Fanuc TP program (LS listing): MAKROSTP.LS

/PROG  MAKROSTP
/ATTR
OWNER		= MNEDITOR;
COMMENT		= "MAKRO_SCHRITT";
PROG_SIZE	= 100704;
CREATE		= DATE 11-01-11  TIME 07:00:00;
MODIFIED	= DATE 18-12-28  TIME 09:20:00;
FILE_NAME	= ;
VERSION		= 0;
LINE_COUNT	= 4405;
MEMORY_SIZE	= 103104;
PROTECT		= READ_WRITE;
TCD:  STACK_SIZE	= 0,
      TASK_PRIORITY	= 100,
      TIME_SLICE	= 0,
      BUSY_LAMP_OFF	= 1,
      ABORT_REQUEST	= 7,
      PAUSE_REQUEST	= 3;
DEFAULT_GROUP	= *,*,*,*,*;
CONTROL_CODE	= 00000000 00000010;
/MN
    :  !Schrittkette Konzernstandard ;
    :  !KS24 ;
    :  !Version: 02 ;
    :  !Stand: 003 MOD KN ;
    :  !letzte Aenderung 30.07.2015 DB ;
    :  !Mod von KN --> S2 mit Wartezeit ;
    :   ;
    :  !Zaehler [41] = aktueller Schritt ;
    :  !Zaehler [42] = letzter Schritt ;
    :  R[41]=0    ;
    :  R[42]=0    ;
    :   ;
    :   ;
    :  !*********************** ;
    :  !*********************** ;
    :  !* Start Makro_Schritt * ;
    :  !*********************** ;
    :  !*********************** ;
    :   ;
    :   ;
    :  !***************************** ;
    :  !*         Schritt 1         * ;
    :  !* E/A's / Flags Ruecksetzen * ;
    :  !***************************** ;
    :   ;
    :  !Loop fuer Schrittkette LBL[1] ;
    :  LBL[1] ;
    :  R[41]=1    ;
    :  !Statusbildschirm einblenden ;
    :  DO[18181]=(OFF) ;
    :  !SK1 KF1 KS1 ;
    :  DO[786]=(OFF) ;
    :  DO[834]=(OFF) ;
    :  DO[842]=(OFF) ;
    :  DO[847]=(OFF) ;
    :  !SK2 KF2 KS2 ;
    :  DO[946]=(OFF) ;
    :  DO[994]=(OFF) ;
    :  DO[995]=(OFF) ;
    :  DO[1002]=(OFF) ;
    :  !SK3 KF3 KS3 ;
    :  DO[1106]=(OFF) ;
    :  DO[1154]=(OFF) ;
    :  DO[1155]=(OFF) ;
    :  DO[1162]=(OFF) ;
    :  !KS1 KS2 KS3 ;
    :  DO[3969]=(OFF) ;
    :  DO[3970]=(OFF) ;
    :  DO[3971]=(OFF) ;
    :  !Auswahl EZ1/SP1 an KF2 ;
    :  F[72]=(OFF) ;
    :  !Auswahl EZ1/SP1 an KF3 ;
    :  F[73]=(OFF) ;
    :  !Auswert. KF Umdrehungen EZ1/SP1 ;
    :  F[94]=(OFF) ;
    :  F[95]=(OFF) ;
    :  F[96]=(OFF) ;
    :  F[97]=(OFF) ;
    :  F[98]=(OFF) ;
    :  F[99]=(OFF) ;
    :  F[100]=(OFF) ;
    :  F[101]=(OFF) ;
    :  F[102]=(OFF) ;
    :  F[103]=(OFF) ;
    :  F[104]=(OFF) ;
    :  F[105]=(OFF) ;
    :  F[106]=(OFF) ;
    :  F[107]=(OFF) ;
    :  F[108]=(OFF) ;
    :  F[109]=(OFF) ;
    :  F[110]=(OFF) ;
    :  F[111]=(OFF) ;
    :  F[112]=(OFF) ;
    :  F[113]=(OFF) ;
    :  F[114]=(OFF) ;
    :  F[115]=(OFF) ;
    :  F[116]=(OFF) ;
    :  F[117]=(OFF) ;
    :  !Auswert. KF Umdrehungen EZ2/SP2 ;
    :  F[150]=(OFF) ;
    :  F[151]=(OFF) ;
    :  F[152]=(OFF) ;
    :  F[153]=(OFF) ;
    :  F[154]=(OFF) ;
    :  F[155]=(OFF) ;
    :  !Auswert. KF Umdrehungen EZ3/SP3 ;
    :  F[186]=(OFF) ;
    :  F[187]=(OFF) ;
    :  F[188]=(OFF) ;
    :  F[189]=(OFF) ;
    :  F[190]=(OFF) ;
    :  F[191]=(OFF) ;
    :  !Hilfsflags beim Fraesen ;
    :  F[287]=(OFF) ;
    :  F[290]=(OFF) ;
    :  F[291]=(OFF) ;
    :  F[301]=(OFF) ;
    :  !Hilfsflags SZ2 an SK1 ;
    :  F[307]=(OFF) ;
    :  F[308]=(OFF) ;
    :  !Hilfsflags KF Initiator ;
    :  F[312]=(OFF) ;
    :  F[313]=(OFF) ;
    :  !RSK Fehlerausgaben ;
    :  F[322]=(OFF) ;
    :  F[323]=(OFF) ;
    :  F[324]=(OFF) ;
    :  F[325]=(OFF) ;
    :  F[326]=(OFF) ;
    :  F[327]=(OFF) ;
    :  F[328]=(OFF) ;
    :  F[329]=(OFF) ;
    :  !Flag KL1 Spueleimer ;
    :  F[352]=(OFF) ;
    :  F[353]=(OFF) ;
    :  !Flag KL2 Spueleimer ;
    :  F[373]=(OFF) ;
    :  F[374]=(OFF) ;
    :  !Flag KL3 Spueleimer ;
    :  F[394]=(OFF) ;
    :  F[395]=(OFF) ;
    :  !Flag MS Reinigung gestartet ;
    :  F[604]=(OFF) ;
    :  F[605]=(OFF) ;
    :  F[608]=(OFF) ;
    :  !Flag für Grundstellung RSK ;
    :  F[321]=(OFF) ;
    :  !Ruecksetzen Fraeszaehler ;
    :  R[1]=0    ;
    :  R[42]=1    ;
    :  JMP LBL[2] ;
    :   ;
    :   ;
    :  !************************ ;
    :  !************************ ;
    :  !* RSK in Grundstellung * ;
    :  !************************ ;
    :  !************************ ;
    :   ;
    :   ;
    :  !*********************** ;
    :  !*      Schritt 2      * ;
    :  !* Funktionsauswertung * ;
    :  !*********************** ;
    :   ;
    :  LBL[2] ;
    :  R[41]=2    ;
    :  F[321]=(ON) ;
    :   ;
    :  !Fraesen ROB EZ1/SP1 SZ1-SZ4 ;
    :  !an KF1 ;
    :  IF ((F[90] AND !F[91]) AND !F[72] AND !F[73] AND (F[64] OR F[65] OR F[66] OR F[67])),R[41]=3 ;
    :   ;
    :  !Fraesen ROB EZ1/SP1 SZ1-SZ4 ;
    :  !an KF2 ;
    :  IF ((F[90] AND !F[91]) AND F[72] AND !F[73] AND (F[64] OR F[65] OR F[66] OR F[67])),R[41]=58 ;
    :   ;
    :  !Fraesen ROB EZ1/SP1 SZ1-SZ4 ;
    :  !an KF3 ;
    :  IF ((F[90] AND !F[91]) AND !F[72] AND F[73] AND (F[64] OR F[65] OR F[66] OR F[67])),R[41]=64 ;
    :   ;
    :  !Fraesen STAT EZ1/SP1 ;
    :  IF (F[92] AND !F[93]),R[41]=9 ;
    :   ;
    :  !Fraesen STAT EZ2/SP2 ;
    :  IF (F[148] AND !F[149]),R[41]=18 ;
    :   ;
    :  !Fraesen STAT EZ3/SP3 ;
    :  IF (F[184] AND !F[185]),R[41]=27 ;
    :   ;
    :  !MS1 Reinigung an KS3 ;
    :  IF (F[603] AND !F[605] AND F[528] AND !F[529]),R[41]=36 ;
    :   ;
    :  !MS2 Reinigung an KS2 ;
    :  IF (F[607] AND !F[609] AND F[528] AND !F[529]),R[41]=40 ;
    :   ;
    :  !KL1 Spueleimer (an Pneum. Schwen ;
    :  !in Arbeitsstellung schwenken ;
    :  IF (!F[352] AND F[353] AND !F[355] AND ((F[523] AND !F[524]) OR (!F[523] AND F[524]))),R[41]=44 ;
    :   ;
    :  !KL1 Spueleimer (an Pneum. Schwen ;
    :  !in Ruhestellung schwenken ;
    :  IF (F[352] AND !F[353] AND !F[355] AND ((F[523] AND !F[524]) OR (!F[523] AND F[524]))),R[41]=45 ;
    :   ;
    :  !KL2 Spueleimer (an Pneum. Schwen ;
    :  !in Arbeitsstellung schwenken ;
    :  IF (!F[373] AND F[374] AND !F[376] AND ((F[523] AND !F[524]) OR (!F[523] AND F[524]))),R[41]=46 ;
    :   ;
    :  !KL2 Spueleimer (an Pneum. Schwen ;
    :  !in Ruhestellung schwenken ;
    :  IF (F[373] AND !F[374] AND !F[376] AND ((F[523] AND !F[524]) OR (!F[523] AND F[524]))),R[41]=47 ;
    :   ;
    :  !KL3 Spueleimer (an Pneum. Schwen ;
    :  !in Arbeitsstellung schwenken ;
    :  IF (!F[394] AND F[395] AND !F[397] AND ((F[523] AND !F[524]) OR (!F[523] AND F[524]))),R[41]=48 ;
    :   ;
    :  !KL3 Spueleimer (an Pneum. Schwen ;
    :  !in Ruhestellung schwenken ;
    :  IF (F[394] AND !F[395] AND !F[397] AND ((F[523] AND !F[524]) OR (!F[523] AND F[524]))),R[41]=49 ;
    :   ;
    :  !MS1 Reinigung (an Pneum. Schwenk ;
    :  IF (F[603] AND !F[605] AND !F[528] AND F[529]),R[41]=50 ;
    :   ;
    :  !Fraesen ROB STP SZ1 ;
    :  IF (F[64] AND !F[65] AND !F[66] AND !F[67] AND F[90] AND !F[91] AND F[565]),R[41]=70 ;
    :   ;
    :  !Wartezeit fuer Synconisation ;
    :  WAIT    .20(sec) ;
    :   ;
    :  R[42]=2    ;
    :  JMP LBL[R[41]] ;
    :   ;
    :   ;
    :  !*************************** ;
    :  !*************************** ;
    :  !* Fraesen Rob EZ1 SZ1-SZ4 * ;
    :  !*          an KF1         * ;
    :  !*************************** ;
    :  !*************************** ;
    :   ;
    :   ;
    :  !**************************** ;
    :  !*        Schritt 3         * ;
    :  !* Rob EZ1 SZ1-SZ4 Auswert. * ;
    :  !**************************** ;
    :   ;
    :  LBL[3] ;
    :  R[41]=3    ;
    :  !RSK gestartet ;
    :  F[321]=(OFF) ;
    :  GO[1]=(31) ;
    :  IF (F[64]),GO[3]=(31) ;
    :  IF (F[65]),GO[3]=(32) ;
    :  IF (F[66]),GO[3]=(33) ;
    :  IF (F[67]),GO[3]=(34) ;
    :  WAIT    .10(sec) ;
    :  DO[116]=(ON) ;
    :  DO[130]=(ON) ;
    :  DO[718]=(OFF) ;
    :  DO[717]=(!DI[717]) ;
    :  DO[18181]=(ON) ;
    :  WAIT (DI[717])    ;
    :  DO[18181]=(OFF) ;
    :  DO[717]=(OFF) ;
    :  !Anwahl Startfraesen ;
    :  IF (F[90] AND F[78] AND !F[79]),R[41]=4 ;
    :  !Anwahl Normalfraesen ;
    :  IF (F[90] AND !F[78] AND F[79]),R[41]=6 ;
    :  R[42]=3    ;
    :  JMP LBL[R[41]] ;
    :   ;
    :  !***************************** ;
    :  !*         Schritt 4         * ;
    :  !* Rob EZ1 SZ1-SZ4 SF Teil 1 * ;
    :  !***************************** ;
    :   ;
    :  LBL[4] ;
    :  R[41]=4    ;
    :  !RSK gestartet ;
    :  F[321]=(OFF) ;
    :  F[329]=(OFF) ;
    :  F[325]=(OFF) ;
    :  DO[718]=(OFF) ;
    :  DO[717]=(!DI[717]) ;
    :  DO[18181]=(ON) ;
    :  WAIT (DI[717])    ;
    :  DO[18181]=(OFF) ;
    :  DO[834]=(ON) ;
    :  DO[858]=(ON) ;
    :  DO[835]=(F[330]) ;
    :  DO[859]=(F[330]) ;
    :  DO[717]=(OFF) ;
    :  !Warte Fraeser laeuft ;
    :  TIMER[7]=((-3)) ;
    :  WAIT ((!DI[834] AND !F[289]) OR (!DI[858] AND F[289]) OR (TIMER[7]>=0))    ;
    :  WAIT ((DI[834] AND !F[289]) OR (DI[858] AND F[289]) OR (TIMER[7]>=0))    ;
    :  F[322]=((TIMER[7]>=0)) ;
    :  DO[18181]=(ON) ;
    :  WAIT ((!DI[834] AND !F[289]) OR (!DI[858] AND F[289]))    ;
    :  WAIT ((DI[834] AND !F[289]) OR (DI[858] AND F[289]))    ;
    :  DO[18181]=(OFF) ;
    :  F[322]=(OFF) ;
    :  !EZ1/SP1 schliessen ;
    :  DO[718]=(ON) ;
    :  TIMER[9]=((-4)) ;
    :  !EZ1/SP1 Kraft erreicht ;
    :  WAIT ((DI[718] AND !DI[772] AND !DI[780] AND !DI[774] AND !DI[775]) OR (TIMER[9]>=0))    ;
    :  DO[18181]=(ON) ;
    :  DO[718]=((TIMER[9]<0)) ;
    :  DO[834]=((TIMER[9]<0)) ;
    :  DO[858]=((TIMER[9]<0)) ;
    :  WAIT ((DI[718] AND !DI[772] AND !DI[780] AND !DI[774] AND !DI[775]) OR DI[26] OR DI[27])    ;
    :  F[325]=(DI[26] OR DI[27]) ;
    :  DO[18181]=(OFF) ;
    :  !EZ1/SP1 Fehler Kraftaufbau ;
    :  IF (F[325]),JMP LBL[406] ;
    :  TIMER[9]=((-5)) ;
    :  LBL[400] ;
    :  WAIT ((!DI[834] AND !F[289]) OR (!DI[858] AND F[289]) OR F[325] OR (TIMER[9]>=0))    ;
    :  WAIT ((DI[834] AND !F[289]) OR (DI[858] AND F[289]) OR F[325] OR (TIMER[9]>=0))    ;
    :  R[1]=(R[1]+1) ;
    :  F[329]=((TIMER[9]>=0)) ;
    :  !Fraeszeit ueberschritten ;
    :  IF (F[329]),JMP LBL[406] ;
    :  IF (F[64]),JMP LBL[402] ;
    :  IF (F[65]),JMP LBL[403] ;
    :  IF (F[66]),JMP LBL[404] ;
    :  IF (F[67]),JMP LBL[405] ;
    :  !Umdrehungen Vergl.SZ1 ;
    :  LBL[402] ;
    :  !Umdrehungen Vergleichen ;
    :  IF (R[1]<R[2]),JMP LBL[400] ;
    :  JMP LBL[401] ;
    :  !Umdrehungen Vergl.SZ2 ;
    :  LBL[403] ;
    :  !Umdrehungen Vergleichen ;
    :  IF (R[1]<R[8]),JMP LBL[400] ;
    :  JMP LBL[401] ;
    :  !Umdrehungen Vergl.SZ3 ;
    :  LBL[404] ;
    :  !Umdrehungen Vergleichen ;
    :  IF (R[1]<R[11]),JMP LBL[400] ;
    :  JMP LBL[401] ;
    :  !Umdrehungen Vergl.SZ4 ;
    :  LBL[405] ;
    :  !Umdrehungen Vergleichen ;
    :  IF (R[1]<R[14]),JMP LBL[400] ;
    :  JMP LBL[401] ;
    :  LBL[401] ;
    :  IF (F[64]),F[94]=(ON) ;
    :  IF (F[65]),F[100]=(ON) ;
    :  IF (F[66]),F[106]=(ON) ;
    :  IF (F[67]),F[112]=(ON) ;
    :  LBL[406] ;
    :  DO[834]=((TIMER[9]<0)) ;
    :  DO[858]=((TIMER[9]<0)) ;
    :  !Fraeser ausblasen EIN ;
    :  DO[835]=(F[330] OR (TIMER[9]<0)) ;
    :  DO[859]=(F[330] OR (TIMER[9]<0)) ;
    :  DO[718]=(OFF) ;
    :  !EZ1/SP1 oeffnen ;
    :  DO[717]=(!DI[717]) ;
    :  DO[18181]=(F[329]) ;
    :  WAIT (!F[329] OR DI[26] OR DI[27])    ;
    :  DO[18181]=(OFF) ;
    :  DO[18181]=(ON) ;
    :  WAIT (DI[717])    ;
    :  DO[18181]=(OFF) ;
    :  DO[717]=(OFF) ;
    :  !Umdrehungen ruecksetzen ;
    :  R[1]=0    ;
    :  R[42]=4    ;
    :  IF (F[329] OR F[325]),JMP LBL[4] ;
    :  JMP LBL[5] ;
    :   ;
    :  !***************************** ;
    :  !*         Schritt 5         * ;
    :  !* Rob EZ1 SZ1-SZ4 SF Teil 2 * ;
    :  !***************************** ;
    :   ;
    :  LBL[5] ;
    :  R[41]=5    ;
    :  !RSK gestartet ;
    :  F[321]=(OFF) ;
    :  F[329]=(OFF) ;
    :  F[325]=(OFF) ;
    :  DO[718]=(OFF) ;
    :  DO[717]=(!DI[717]) ;
    :  DO[18181]=(ON) ;
    :  WAIT (DI[717])    ;
    :  DO[18181]=(OFF) ;
    :  DO[834]=(ON) ;
    :  DO[858]=(ON) ;
    :  DO[717]=(OFF) ;
    :  !EZ1/SP1 schliessen ;
    :  DO[718]=(ON) ;
    :  !Fraeser ausblasen AUS/AN ;
    :  DO[835]=(F[330]) ;
    :  DO[859]=(F[330]) ;
    :  TIMER[9]=((-4)) ;
    :  !EZ1/SP1 Kraft erreicht ;
    :  WAIT ((DI[718] AND !DI[772] AND !DI[780] AND !DI[774] AND !DI[775]) OR (TIMER[9]>=0))    ;
    :  DO[18181]=(ON) ;
    :  DO[718]=((TIMER[9]<0)) ;
    :  DO[834]=((TIMER[9]<0)) ;
    :  DO[858]=((TIMER[9]<0)) ;
    :  WAIT ((DI[718] AND !DI[772] AND !DI[780] AND !DI[774] AND !DI[775]) OR DI[26] OR DI[27])    ;
    :  F[325]=(DI[26] OR DI[27]) ;
    :  DO[18181]=(OFF) ;
    :  !EZ1/SP1 Fehler Kraftaufbau ;
    :  IF (F[325]),JMP LBL[5] ;
    :  TIMER[9]=((-5)) ;
    :  LBL[500] ;
    :  WAIT ((!DI[834] AND !F[289]) OR (!DI[858] AND F[289]) OR F[325] OR (TIMER[9]>=0))    ;
    :  WAIT ((DI[834] AND !F[289]) OR (DI[858] AND F[289]) OR F[325] OR (TIMER[9]>=0))    ;
    :  R[1]=(R[1]+1) ;
    :  F[329]=((TIMER[9]>=0)) ;
    :  !Fraeszeit ueberschritten ;
    :  IF (F[329]),JMP LBL[506] ;
    :  IF (F[64]),JMP LBL[502] ;
    :  IF (F[65]),JMP LBL[503] ;
    :  IF (F[66]),JMP LBL[504] ;
    :  IF (F[67]),JMP LBL[505] ;
    :  !Umdrehungen Vergl.SZ1 ;
    :  LBL[502] ;
    :  !Umdrehungen Vergleichen ;
    :  IF (R[1]<R[3]),JMP LBL[500] ;
    :  JMP LBL[501] ;
    :  !Umdrehungen Vergl.SZ2 ;
    :  LBL[503] ;
    :  !Umdrehungen Vergleichen ;
    :  IF (R[1]<R[9]),JMP LBL[500] ;
    :  JMP LBL[501] ;
    :  !Umdrehungen Vergl.SZ3 ;
    :  LBL[504] ;
    :  !Umdrehungen Vergleichen ;
    :  IF (R[1]<R[12]),JMP LBL[500] ;
    :  JMP LBL[501] ;
    :  !Umdrehungen Vergl.SZ4 ;
    :  LBL[505] ;
    :  !Umdrehungen Vergleichen ;
    :  IF (R[1]<R[15]),JMP LBL[500] ;
    :  JMP LBL[501] ;
    :  LBL[501] ;
    :  IF (F[64]),F[96]=(ON) ;
    :  IF (F[65]),F[102]=(ON) ;
    :  IF (F[66]),F[108]=(ON) ;
    :  IF (F[67]),F[114]=(ON) ;
    :  LBL[506] ;
    :  DO[834]=((TIMER[9]<0)) ;
    :  DO[858]=((TIMER[9]<0)) ;
    :  !Fraeser ausblasen EIN ;
    :  DO[835]=PULSE,4.0sec ;
    :  DO[859]=PULSE,4.0sec ;
    :  DO[718]=(OFF) ;
    :  !EZ1/SP1 oeffnen ;
    :  DO[717]=(!DI[717]) ;
    :  DO[18181]=(F[329]) ;
    :  WAIT (!F[329] OR DI[26] OR DI[27])    ;
    :  DO[18181]=(OFF) ;
    :  DO[18181]=(ON) ;
    :  WAIT (DI[717])    ;
    :  DO[18181]=(OFF) ;
    :  DO[717]=(OFF) ;
    :  !Umdrehungen ruecksetzen ;
    :  R[1]=0    ;
    :  R[42]=5    ;
    :  IF (F[329] OR F[325]),JMP LBL[5] ;
    :  JMP LBL[7] ;
    :   ;
    :  !********************** ;
    :  !*     Schritt 6      * ;
    :  !* Rob EZ1 SZ1-SZ4 NF * ;
    :  !********************** ;
    :   ;
    :  LBL[6] ;
    :  R[41]=6    ;
    :  !RSK gestartet ;
    :  F[321]=(OFF) ;
    :  F[329]=(OFF) ;
    :  F[325]=(OFF) ;
    :  !Zähler wegspeichern für 2ten Hub ;
    :  R[45]=R[4]    ;
    :  IF (F[98] AND F[732]),R[4]=R[43] ;
    :  !Überprüfungung Zangenstellung ;
    :  DO[718]=(OFF) ;
    :  DO[717]=(!DI[717]) ;
    :  DO[18181]=(ON) ;
    :  WAIT (DI[717])    ;
    :  DO[18181]=(OFF) ;
    :  DO[834]=(ON) ;
    :  DO[835]=(F[330]) ;
    :  DO[858]=(ON) ;
    :  DO[859]=(F[330]) ;
    :  DO[717]=(OFF) ;
    :  !Warte Fraeser laeuft ;
    :  TIMER[7]=((-3)) ;
    :  WAIT ((!DI[834] AND !F[289]) OR (!DI[858] AND F[289]) OR (TIMER[7]>=0))    ;
    :  WAIT ((DI[834] AND !F[289]) OR (DI[858] AND F[289]) OR (TIMER[7]>=0))    ;
    :  F[322]=((TIMER[7]>=0)) ;
    :  DO[18181]=(ON) ;
    :  WAIT ((!DI[834] AND !F[289]) OR (!DI[858] AND F[289]))    ;
    :  WAIT ((DI[834] AND !F[289]) OR (DI[858] AND F[289]))    ;
    :  DO[18181]=(OFF) ;
    :  F[322]=(OFF) ;
    :  !EZ1/SP1 schliessen ;
    :  DO[718]=(ON) ;
    :  TIMER[9]=((-4)) ;
    :  !EZ1/SP1 Kraft erreicht ;
    :  WAIT ((DI[718] AND !DI[772] AND !DI[780] AND !DI[774] AND !DI[775]) OR (TIMER[9]>=0))    ;
    :  DO[18181]=(ON) ;
    :  DO[718]=((TIMER[9]<0)) ;
    :  DO[834]=((TIMER[9]<0)) ;
    :  DO[858]=((TIMER[9]<0)) ;
    :  WAIT ((DI[718] AND !DI[772] AND !DI[780] AND !DI[774] AND !DI[775]) OR DI[26] OR DI[27])    ;
    :  F[325]=(DI[26] OR DI[27]) ;
    :  DO[18181]=(OFF) ;
    :  !EZ1/SP1 Fehler Kraftaufbau ;
    :  IF (F[325]),JMP LBL[6] ;
    :  TIMER[9]=((-5)) ;
    :  LBL[600] ;
    :  WAIT ((!DI[834] AND !F[289]) OR (!DI[858] AND F[289]) OR F[325] OR (TIMER[9]>=0))    ;
    :  WAIT ((DI[834] AND !F[289]) OR (DI[858] AND F[289]) OR F[325] OR (TIMER[9]>=0))    ;
    :  R[1]=(R[1]+1) ;
    :  F[329]=((TIMER[9]>=0)) ;
    :  !Fraeszeit ueberschritten ;
    :  IF (F[329]),JMP LBL[606] ;
    :  IF (F[64]),JMP LBL[602] ;
    :  IF (F[65]),JMP LBL[603] ;
    :  IF (F[66]),JMP LBL[604] ;
    :  IF (F[67]),JMP LBL[605] ;
    :  !Umdrehungen Vergl.SZ1 ;
    :  LBL[602] ;
    :  !Umdrehungen Vergleichen ;
    :  IF (R[1]<R[4]),JMP LBL[600] ;
    :  JMP LBL[601] ;
    :  !Umdrehungen Vergl.SZ2 ;
    :  LBL[603] ;
    :  !Umdrehungen Vergleichen ;
    :  IF (R[1]<R[10]),JMP LBL[600] ;
    :  !Umdrehungen Vergl.SZ3 ;
    :  LBL[604] ;
    :  !Umdrehungen Vergleichen ;
    :  IF (R[1]<R[13]),JMP LBL[600] ;
    :  JMP LBL[601] ;
    :  !Umdrehungen Vergl.SZ4 ;
    :  LBL[605] ;
    :  !Umdrehungen Vergleichen ;
    :  IF (R[1]<R[16]),JMP LBL[600] ;
    :  LBL[601] ;
    :  !EZ1/SP1 2 Huebe bei NF ;
    :  IF (!F[130]),JMP LBL[606] ;
    :  IF (F[98]),F[96]=(ON) ;
    :  IF (F[104]),F[96]=(ON) ;
    :  IF (F[110]),F[96]=(ON) ;
    :  IF (F[116]),F[96]=(ON) ;
    :  IF (F[64]),F[98]=(ON) ;
    :  IF (F[65]),F[104]=(ON) ;
    :  IF (F[66]),F[110]=(ON) ;
    :  IF (F[67]),F[116]=(ON) ;
    :  LBL[606] ;
    :  DO[834]=((TIMER[9]<0)) ;
    :  DO[858]=((TIMER[9]<0)) ;
    :  !Fraeser ausblasen EIN ;
    :  DO[835]=PULSE,4.0sec ;
    :  DO[859]=PULSE,4.0sec ;
    :  DO[718]=(OFF) ;
    :  !EZ1/SP1 oeffnen ;
    :  DO[717]=(!DI[717]) ;
    :  DO[18181]=(F[329]) ;
    :  WAIT (!F[329] OR DI[26] OR DI[27])    ;
    :  DO[18181]=(OFF) ;
    :  DO[18181]=(ON) ;
    :  WAIT (DI[717])    ;
    :  DO[18181]=(OFF) ;
    :  DO[717]=(OFF) ;
    :  !Umdrehungen ruecksetzen ;
    :  R[1]=0    ;
    :  R[42]=6    ;
    :  !Zähler umschreiben für 2ten Hub ;
    :  IF (F[98] AND F[732] AND F[64]),GO[3]=36 ;
    :  IF (F[104] AND F[732] AND F[65]),GO[3]=37 ;
    :  IF (F[110] AND F[732] AND F[66]),GO[3]=38 ;
    :  IF (F[116] AND F[732] AND F[67]),GO[3]=39 ;
    :  IF (F[96] AND F[732]),R[4]=R[45] ;
    :  !Aufruf 2ter Hub ;
    :  IF (F[329] OR (!F[96] AND F[130])),JMP LBL[6] ;
    :  IF (F[64]),F[98]=(ON) ;
    :  IF (F[65]),F[104]=(ON) ;
    :  IF (F[66]),F[110]=(ON) ;
    :  IF (F[67]),F[116]=(ON) ;
    :  JMP LBL[7] ;
    :   ;
    :  !******************************* ;
    :  !*         Schritt 7           * ;
    :  !* Rob EZ1 SZ1-SZ4 i.O./n.i.O. * ;
    :  !******************************* ;
    :   ;
    :  LBL[7] ;
    :  R[41]=7    ;
    :  !Fraesueberwachung starten ;
    :  IF (F[64]),JMP LBL[701] ;
    :  IF (F[65]),JMP LBL[702] ;
    :  IF (F[66]),JMP LBL[703] ;
    :  IF (F[67]),JMP LBL[704] ;
    :  LBL[701] ;
    :  TIMER[7]=((-3)) ;
    :  WAIT (F[64] AND ((F[79] AND F[98]) OR (F[78] AND F[94] AND F[96])) OR (TIMER[7]>=0))    ;
    :  F[329]=((TIMER[7]>=0)) ;
    :  DO[18181]=(ON) ;
    :  WAIT (F[64] AND ((F[79] AND F[98]) OR (F[78] AND F[94] AND F[96])))    ;
    :  DO[18181]=(OFF) ;
    :  JMP LBL[700] ;
    :  LBL[702] ;
    :  TIMER[7]=((-3)) ;
    :  WAIT (F[65] AND ((F[79] AND F[104]) OR (F[78] AND F[100] AND F[102])) OR (TIMER[7]>=0))    ;
    :  F[329]=((TIMER[7]>=0)) ;
    :  DO[18181]=(ON) ;
    :  WAIT (F[65] AND ((F[79] AND F[104]) OR (F[78] AND F[100] AND F[102])))    ;
    :  DO[18181]=(OFF) ;
    :  JMP LBL[700] ;
    :  LBL[703] ;
    :  TIMER[7]=((-3)) ;
    :  WAIT (F[66] AND ((F[79] AND F[110]) OR (F[78] AND F[106] AND F[108])) OR (TIMER[7]>=0))    ;
    :  F[329]=((TIMER[7]>=0)) ;
    :  DO[18181]=(ON) ;
    :  WAIT (F[66] AND ((F[79] AND F[110]) OR (F[78] AND F[106] AND F[108])))    ;
    :  DO[18181]=(OFF) ;
    :  JMP LBL[700] ;
    :  LBL[704] ;
    :  TIMER[7]=((-3)) ;
    :  WAIT (F[67] AND ((F[79] AND F[116]) OR (F[78] AND F[112] AND F[114])) OR (TIMER[7]>=0))    ;
    :  F[329]=((TIMER[7]>=0)) ;
    :  DO[18181]=(ON) ;
    :  WAIT (F[67] AND ((F[79] AND F[116]) OR (F[78] AND F[112] AND F[114])))    ;
    :  DO[18181]=(OFF) ;
    :  JMP LBL[700] ;
    :  LBL[700] ;
    :  R[41]=8    ;
    :  !KF1 U-Merker ruecksetzen ;
    :  F[94]=(OFF) ;
    :  F[96]=(OFF) ;
    :  F[98]=(OFF) ;
    :  F[100]=(OFF) ;
    :  F[102]=(OFF) ;
    :  F[104]=(OFF) ;
    :  F[106]=(OFF) ;
    :  F[108]=(OFF) ;
    :  F[110]=(OFF) ;
    :  F[112]=(OFF) ;
    :  F[114]=(OFF) ;
    :  F[116]=(OFF) ;
    :  R[42]=7    ;
    :  JMP LBL[R[41]] ;
    :   ;
    :  !***************************** ;
    :  !*        Schritt 8          * ;
    :  !* Rob EZ1 SZ1-SZ4 Quitt SK1 * ;
    :  !***************************** ;
    :   ;
    :  LBL[8] ;
    :  R[41]=8    ;
    :  !RSK gestartet ;
    :  F[321]=(OFF) ;
    :  IF (F[64]),GO[3]=1 ;
    :  IF (F[65]),GO[3]=2 ;
    :  IF (F[66]),GO[3]=3 ;
    :  IF (F[67]),GO[3]=4 ;
    :  WAIT    .10(sec) ;
    :  DO[786]=(ON) ;
    :  DO[116]=(OFF) ;
    :  DO[130]=(OFF) ;
    :  DO[18181]=(ON) ;
    :  WAIT (!DI[786] AND DI[787] AND !DI[788])    ;
    :  !FK Fraesen ;
    :  F[91]=(!F[329]) ;
    :  DO[18181]=(OFF) ;
    :  DO[786]=(OFF) ;
    :  R[42]=8    ;
    :  JMP LBL[1] ;
    :   ;
    :   ;
    :  !************************ ;
    :  !************************ ;
    :  !* Fraesen STAT EZ1/SP1 * ;
    :  !************************ ;
    :  !************************ ;
    :   ;
    :   ;
    :  !****************************** ;
    :  !*         Schritt 9          * ;
    :  !*        STAT EZ1/SP1        * ;
    :  !* KS1 in Arbeitsst.schwenken * ;
    :  !****************************** ;
    :   ;
    :  LBL[9] ;
    :  R[41]=9    ;
    :  !RSK gestartet ;
    :  F[321]=(OFF) ;
    :  GO[1]=(31) ;
    :  GO[3]=(31) ;
    :  WAIT    .10(sec) ;
    :  DO[758]=(F[78]) ;
    :  DO[759]=(F[79]) ;
    :  DO[116]=(ON) ;
    :  DO[130]=(ON) ;
    :  DO[718]=(OFF) ;
    :  DO[717]=(!DI[717]) ;
    :  DO[18181]=(ON) ;
    :  WAIT (DI[717])    ;
    :  DO[18181]=(OFF) ;
    :  DO[717]=(OFF) ;
    :  !Ueberwachungszeit Grundstellung ;
    :  TIMER[8]=((-4)) ;
    :  WAIT ((DI[842] AND !DI[843] AND !DI[844] AND DI[845]) OR (TIMER[8]>=0))    ;
    :  F[323]=((TIMER[8]>=0)) ;
    :  DO[18181]=((TIMER[8]>=0)) ;
    :  WAIT (DI[842] AND !DI[843] AND !DI[844] AND DI[845])    ;
    :  DO[18181]=(OFF) ;
    :  F[323]=(OFF) ;
    :  TIMER[8]=((-4)) ;
    :  DO[835]=(F[564]) ;
    :  WAIT ((DI[835] AND F[564]) OR (!DI[835] AND !F[564]) OR (TIMER[8]>=0))    ;
    :  F[323]=((TIMER[8]>=0)) ;
    :  DO[18181]=((TIMER[8]>=0)) ;
    :  WAIT ((DI[835] AND F[564]) OR (!DI[835] AND !F[564]))    ;
    :  DO[18181]=(OFF) ;
    :  F[323]=(OFF) ;
    :  !Ueberwachungszeit KS1 Schwenken ;
    :  TIMER[8]=((-6)) ;
    :  !KS1 in Arbeitst. schwenken ;
    :  DO[3972]=(ON) ;
    :  WAIT (DI[841] OR (TIMER[8]>=0))    ;
    :  DO[18181]=((TIMER[8]>=0)) ;
    :  WAIT (DI[841])    ;
    :  TIMER[8]=((-6)) ;
    :  DO[18181]=(OFF) ;
    :  WAIT ((!DI[842] AND DI[843] AND DI[844] AND !DI[845]) OR (TIMER[8]>=0))    ;
    :  F[324]=((TIMER[8]>=0)) ;
    :  DO[3972]=(OFF) ;
    :  DO[18181]=((TIMER[8]>=0)) ;
    :  WAIT ((!DI[842] AND DI[843] AND DI[844] AND !DI[845]) OR DI[26])    ;
    :  DO[18181]=(OFF) ;
    :  F[324]=(OFF) ;
    :  !Sprung zurueck bei KS1 Fehler ;
    :  IF (TIMER[8]>=0),JMP LBL[9] ;
    :  DO[835]=(OFF) ;
    :  TIMER[11]=((R[24])) ;
    :  WAIT ((TIMER[11]>=0) OR !F[564])    ;
    :  TIMER[11]=STOP ;
    :  DO[18181]=(ON) ;
    :  WAIT ((F[92] AND F[78]) OR (F[92] AND F[79]))    ;
    :  DO[18181]=(OFF) ;
    :  !Anwahl Startfraesen ;
    :  IF (!DI[842] AND DI[843] AND F[92] AND F[78] AND !F[301]),R[41]=10 ;
    :  !Anwahl Normalfraesen ;
    :  IF (!DI[842] AND DI[843] AND F[92] AND (F[79] OR F[301])),R[41]=12 ;
    :  R[42]=9    ;
    :  JMP LBL[R[41]] ;
    :   ;
    :  !************************** ;
    :  !*       Schritt 10       * ;
    :  !* STAT EZ1/SP1 SF Teil 1 * ;
    :  !************************** ;
    :   ;
    :  LBL[10] ;
    :  R[41]=10    ;
    :  !RSK gestartet ;
    :  F[321]=(OFF) ;
    :  F[329]=(OFF) ;
    :  F[325]=(OFF) ;
    :  DO[718]=(OFF) ;
    :  DO[717]=(!DI[717]) ;
    :  DO[18181]=(ON) ;
    :  WAIT (DI[717])    ;
    :  DO[717]=(OFF) ;
    :  DO[18181]=(OFF) ;
    :  DO[834]=(ON) ;
    :  !Warte Fraeser laeuft ;
    :  TIMER[7]=((-3)) ;
    :  WAIT (!DI[834] OR (TIMER[7]>=0))    ;
    :  WAIT (DI[834] OR (TIMER[7]>=0))    ;
    :  F[322]=((TIMER[7]>=0)) ;
    :  DO[18181]=(ON) ;
    :  WAIT (!DI[834])    ;
    :  WAIT (DI[834])    ;
    :  DO[18181]=(OFF) ;
    :  F[322]=(OFF) ;
    :  !EZ1/SP1 schliessen ;
    :  DO[718]=(ON) ;
    :  !Fraeser ausblasen AUS/EIN ;
    :  DO[847]=(F[330]) ;
    :  TIMER[9]=((-4)) ;
    :  !EZ1/SP1 Kraft erreicht ;
    :  WAIT ((DI[718] AND !DI[772] AND !DI[780] AND !DI[774] AND !DI[775]) OR (TIMER[9]>=0))    ;
    :  F[325]=((TIMER[9]>=0)) ;
    :  DO[18181]=(ON) ;
    :  DO[718]=((TIMER[9]<0)) ;
    :  DO[834]=((TIMER[9]<0)) ;
    :  WAIT ((DI[718] AND !DI[772] AND !DI[780] AND !DI[774] AND !DI[775]) OR DI[26] OR DI[27])    ;
    :  DO[18181]=(OFF) ;
    :  !EZ1/SP1 Fehler Kraftaufbau ;
    :  IF (F[325]),JMP LBL[1001] ;
    :  TIMER[9]=((-5)) ;
    :  LBL[1000] ;
    :  WAIT (!DI[834] OR F[325] OR (TIMER[9]>=0))    ;
    :  WAIT (DI[834] OR F[325] OR (TIMER[9]>=0))    ;
    :  R[1]=(R[1]+1) ;
    :  F[329]=((TIMER[9]>=0)) ;
    :  !Fraeszeit ueberschritten ;
    :  IF (F[329]),JMP LBL[1001] ;
    :  !Umdrehungen Vergleichen ;
    :  IF (R[1]<R[2]),JMP LBL[1000] ;
    :  F[94]=(ON) ;
    :  LBL[1001] ;
    :  DO[834]=((TIMER[9]<0)) ;
    :  !Fraeser ausblasen EIN ;
    :  DO[847]=(F[330] OR (TIMER[9]<0)) ;
    :  DO[718]=(OFF) ;
    :  !EZ1/SP1 oeffnen ;
    :  DO[717]=(!DI[717]) ;
    :  DO[18181]=(F[329]) ;
    :  WAIT (!F[329] OR DI[26] OR DI[27])    ;
    :  DO[18181]=(OFF) ;
    :  DO[18181]=(ON) ;
    :  WAIT (DI[717])    ;
    :  DO[18181]=(OFF) ;
    :  DO[717]=(OFF) ;
    :  !Umdrehungen ruecksetzen ;
    :  R[1]=0    ;
    :  R[42]=10    ;
    :  IF (F[329] OR F[325]),JMP LBL[10] ;
    :  JMP LBL[11] ;
    :   ;
    :  !************************** ;
    :  !*       Schritt 11       * ;
    :  !* STAT EZ1/SP1 SF Teil 2 * ;
    :  !************************** ;
    :   ;
    :  LBL[11] ;
    :  R[41]=11    ;
    :  !RSK gestartet ;
    :  F[321]=(OFF) ;
    :  F[329]=(OFF) ;
    :  F[325]=(OFF) ;
    :  DO[718]=(OFF) ;
    :  DO[717]=(!DI[717]) ;
    :  DO[18181]=(ON) ;
    :  WAIT (DI[717])    ;
    :  DO[18181]=(OFF) ;
    :  DO[834]=(ON) ;
    :  DO[717]=(OFF) ;
    :  !EZ1/SP1 schliessen ;
    :  DO[718]=(ON) ;
    :  !Fraeser ausblasen AUS/EIN ;
    :  DO[847]=(F[330]) ;
    :  TIMER[9]=((-4)) ;
    :  !EZ1/SP1 Kraft erreicht ;
    :  WAIT ((DI[718] AND !DI[772] AND !DI[780] AND !DI[774] AND !DI[775]) OR (TIMER[9]>=0))    ;
    :  F[325]=((TIMER[9]>=0)) ;
    :  DO[18181]=(ON) ;
    :  DO[718]=((TIMER[9]<0)) ;
    :  DO[834]=((TIMER[9]<0)) ;
    :  WAIT ((DI[718] AND !DI[772] AND !DI[780] AND !DI[774] AND !DI[775]) OR DI[26] OR DI[27])    ;
    :  DO[18181]=(OFF) ;
    :  !EZ1/SP1 Fehler Kraftaufbau ;
    :  IF (F[325]),JMP LBL[1101] ;
    :  TIMER[9]=((-5)) ;
    :  LBL[1100] ;
    :  WAIT (!DI[834] OR F[325] OR (TIMER[9]>=0))    ;
    :  WAIT (DI[834] OR F[325] OR (TIMER[9]>=0))    ;
    :  R[1]=(R[1]+1) ;
    :  F[329]=((TIMER[9]>=0)) ;
    :  !Fraeszeit ueberschritten ;
    :  IF (F[329]),JMP LBL[1101] ;
    :  !Umdrehungen Vergleichen ;
    :  IF (R[1]<R[3]),JMP LBL[1100] ;
    :  F[96]=(ON) ;
    :  LBL[1101] ;
    :  DO[834]=((TIMER[9]<0)) ;
    :  !Fraeser ausblasen EIN ;
    :  DO[847]=PULSE,4.0sec ;
    :  DO[718]=(OFF) ;
    :  !EZ1/SP1 oeffnen ;
    :  DO[717]=(!DI[717]) ;
    :  DO[18181]=(F[329]) ;
    :  WAIT (!F[329] OR DI[26] OR DI[27])    ;
    :  DO[18181]=(OFF) ;
    :  DO[18181]=(ON) ;
    :  WAIT (DI[717])    ;
    :  DO[18181]=(OFF) ;
    :  DO[717]=(OFF) ;
    :  !Umdrehungen ruecksetzen ;
    :  R[1]=0    ;
    :  R[42]=11    ;
    :  IF (F[329] OR F[325]),JMP LBL[11] ;
    :  JMP LBL[13] ;
    :   ;
    :  !******************* ;
    :  !*   Schritt 12    * ;
    :  !* STAT EZ1/SP1 NF * ;
    :  !******************* ;
    :   ;
    :  LBL[12] ;
    :  R[41]=12    ;
    :  !RSK gestartet ;
    :  F[321]=(OFF) ;
    :  F[329]=(OFF) ;
    :  F[325]=(OFF) ;
    :  !Zähler wegspeichern für 2ten Hub ;
    :  R[45]=R[4]    ;
    :  IF (F[98] AND F[732]),R[4]=R[43] ;
    :  !Überprüfungung Zangenstellung ;
    :  DO[718]=(OFF) ;
    :  DO[717]=(!DI[717]) ;
    :  DO[18181]=(ON) ;
    :  WAIT (DI[717])    ;
    :  DO[18181]=(OFF) ;
    :  DO[834]=(ON) ;
    :  DO[717]=(OFF) ;
    :  !EZ1/SP1 schliessen ;
    :  DO[718]=(ON) ;
    :  !Fraeser ausblasen AUS/EIN ;
    :  DO[847]=(F[330]) ;
    :  TIMER[9]=((-4)) ;
    :  !EZ1/SP1 Kraft erreicht ;
    :  WAIT ((DI[718] AND !DI[772] AND !DI[780] AND !DI[774] AND !DI[775]) OR (TIMER[9]>=0))    ;
    :  F[325]=((TIMER[9]>=0)) ;
    :  DO[18181]=(ON) ;
    :  DO[718]=((TIMER[9]<0)) ;
    :  DO[834]=((TIMER[9]<0)) ;
    :  WAIT ((DI[718] AND !DI[772] AND !DI[780] AND !DI[774] AND !DI[775]) OR DI[26] OR DI[27])    ;
    :  DO[18181]=(OFF) ;
    :  !EZ1/SP1 Fehler Kraftaufbau ;
    :  IF (F[325]),JMP LBL[1201] ;
    :  TIMER[9]=((-5)) ;
    :  LBL[1200] ;
    :  WAIT (!DI[834] OR F[325] OR (TIMER[9]>=0))    ;
    :  WAIT (DI[834] OR F[325] OR (TIMER[9]>=0))    ;
    :  R[1]=(R[1]+1) ;
    :  F[329]=((TIMER[9]>=0)) ;
    :  !Fraeszeit ueberschritten ;
    :  IF (F[329]),JMP LBL[1201] ;
    :  !Umdrehungen Vergleichen ;
    :  IF (R[1]<R[4]),JMP LBL[1200] ;
    :  !EZ1/SP1 2 Huebe bei NF ;
    :  IF (!F[130]),JMP LBL[1201] ;
    :  IF (F[98]),F[96]=(ON) ;
    :  F[98]=(ON) ;
    :  LBL[1201] ;
    :  DO[834]=((TIMER[9]<0)) ;
    :  !Fraeser ausblasen EIN ;
    :  DO[847]=PULSE,4.0sec ;
    :  !EZ1/SP1 oeffnen ;
    :  DO[718]=(OFF) ;
    :  DO[717]=(!DI[717]) ;
    :  DO[18181]=(F[329]) ;
    :  WAIT (!F[329] OR DI[26] OR DI[27])    ;
    :  DO[18181]=(OFF) ;
    :  DO[18181]=(ON) ;
    :  WAIT (DI[717])    ;
    :  DO[18181]=(OFF) ;
    :  DO[717]=(OFF) ;
    :  !Umdrehungen ruecksetzen ;
    :  R[1]=0    ;
    :  R[42]=12    ;
    :  !Zähler umschreiben für 2ten Hub ;
    :  IF (F[98] AND F[732]),GO[3]=36 ;
    :  IF (F[96] AND F[732]),R[4]=R[45] ;
    :  IF (F[329] OR F[325] OR (!F[96] AND F[130])),JMP LBL[12] ;
    :  F[98]=(ON) ;
    :  JMP LBL[13] ;
    :   ;
    :  !**************************** ;
    :  !*        Schritt 13        * ;
    :  !* STAT EZ1/SP1 i.O./n.i.O. * ;
    :  !**************************** ;
    :   ;
    :  LBL[13] ;
    :  R[41]=13    ;
    :  !Fraesueberwachung starten ;
    :  TIMER[7]=((-5)) ;
    :  WAIT ((F[78] OR F[79]) AND (F[98] OR (F[94] AND F[96])) OR (TIMER[7]>=0))    ;
    :  F[329]=((TIMER[7]>=0)) ;
    :  IF (!F[329]),R[41]=14 ;
    :  IF (F[329]),R[41]=12 ;
    :  !KF1 U-Merker ruecksetzen ;
    :  F[94]=(OFF) ;
    :  F[96]=(OFF) ;
    :  F[98]=(OFF) ;
    :  R[42]=13    ;
    :  JMP LBL[R[41]] ;
    :   ;
    :  !*************************** ;
    :  !*       Schritt 14        * ;
    :  !*    STAT EZ1/SP1 KS1     * ;
    :  !* KS1 in Ruhest.schwenken * ;
    :  !*************************** ;
    :   ;
    :  LBL[14] ;
    :  R[41]=14    ;
    :  !RSK gestartet ;
    :  F[321]=(OFF) ;
    :  DO[718]=(OFF) ;
    :  DO[717]=(!DI[717]) ;
    :  DO[18181]=(ON) ;
    :  WAIT (DI[717])    ;
    :  DO[18181]=(OFF) ;
    :  DO[717]=(OFF) ;
    :  TIMER[8]=((-4)) ;
    :  WAIT ((DI[844] AND !DI[842] AND !DI[845] AND DI[843]) OR (TIMER[8]>=0))    ;
    :  F[324]=((TIMER[8]>=0)) ;
    :  DO[18181]=((TIMER[8]>=0)) ;
    :  WAIT (DI[844] AND !DI[842] AND !DI[845] AND DI[843])    ;
    :  DO[18181]=(OFF) ;
    :  F[324]=(OFF) ;
    :  TIMER[8]=((-4)) ;
    :  DO[835]=(F[564]) ;
    :  WAIT ((DI[835] AND F[564]) OR (!DI[835] AND !F[564]) OR (TIMER[8]>=0))    ;
    :  F[323]=((TIMER[8]>=0)) ;
    :  DO[18181]=((TIMER[8]>=0)) ;
    :  WAIT ((DI[835] AND F[564]) OR (!DI[835] AND !F[564]))    ;
    :  DO[18181]=(OFF) ;
    :  F[323]=(OFF) ;
    :  !Ueberwachungszeit KS1 Schwenken ;
    :  TIMER[8]=((-4)) ;
    :  DO[3969]=(ON) ;
    :  WAIT (DI[841] OR (TIMER[8]>=0))    ;
    :  DO[18181]=((TIMER[8]>=0)) ;
    :  WAIT (DI[841])    ;
    :  DO[18181]=(OFF) ;
    :  TIMER[8]=((-6)) ;
    :  WAIT ((!DI[844] AND DI[842] AND DI[845] AND !DI[843]) OR (TIMER[8]>=0))    ;
    :  F[323]=((TIMER[8]>=0)) ;
    :  DO[3969]=(OFF) ;
    :  DO[18181]=((TIMER[8]>=0)) ;
    :  WAIT ((!DI[844] AND DI[842] AND DI[845] AND !DI[843]) OR DI[26])    ;
    :  DO[18181]=(OFF) ;
    :  DO[835]=(OFF) ;
    :  F[323]=(OFF) ;
    :  DO[834]=(OFF) ;
    :  !Sprung zurueck bei KS1 Fehler ;
    :  IF (TIMER[8]>=0),JMP LBL[14] ;
    :  R[42]=14    ;
    :  JMP LBL[15] ;
    :   ;
    :  !*********************** ;
    :  !*     Schritt 15      * ;
    :  !*    STAT EZ1/SP1     * ;
    :  !* Messen nach Fraesen * ;
    :  !*********************** ;
    :   ;
    :  LBL[15] ;
    :  R[41]=15    ;
    :  !RSK gestartet ;
    :  F[321]=(OFF) ;
    :  GO[3]=1 ;
    :  WAIT    .10(sec) ;
    :  DO[786]=(ON) ;
    :  DO[18181]=(ON) ;
    :  WAIT (!DI[786] AND DI[787] AND !DI[788])    ;
    :  DO[18181]=(OFF) ;
    :  DO[786]=(OFF) ;
    :  GO[1]=(31) ;
    :  GO[3]=(31) ;
    :  WAIT    .10(sec) ;
    :  DO[757]=(ON) ;
    :  TIMER[9]=((-8)) ;
    :  WAIT (DI[757] OR (TIMER[9]>=0))    ;
    :  F[326]=((TIMER[9]>=0)) ;
    :  DO[18181]=(ON) ;
    :  WAIT (DI[757] OR DI[26] OR DI[27])    ;
    :  DO[18181]=(OFF) ;
    :  F[326]=(OFF) ;
    :  F[85]=(DI[776] OR DI[777]) ;
    :  DO[757]=(OFF) ;
    :  F[86]=(DI[736] OR (DI[735] AND DI[734] AND DI[733])) ;
    :  TIMER[7]=((-2)) ;
    :  WAIT ((!F[85] AND !F[86]) OR (TIMER[7]>=0))    ;
    :  F[329]=((TIMER[7]>=0)) ;
    :  DO[18181]=(F[329]) ;
    :  WAIT ((!F[85] AND !F[86]) OR DI[26] OR DI[27])    ;
    :  DO[18181]=(OFF) ;
    :  F[329]=(OFF) ;
    :  F[298]=(F[85] OR F[86]) ;
    :  DO[717]=(!DI[717]) ;
    :  DO[18181]=(ON) ;
    :  WAIT ((DI[717] AND !DI[784]) OR (DI[717] AND F[298]))    ;
    :  DO[18181]=(OFF) ;
    :  DO[717]=(OFF) ;
    :  R[42]=15    ;
    :  !EZ1/SP1 wiederh. bei Messfehler ;
    :  IF (DI[777]),JMP LBL[17] ;
    :  DO[758]=(OFF) ;
    :  DO[759]=(OFF) ;
    :  !KS nicht bei K-Verschleiss ;
    :  IF (F[298]),JMP LBL[9] ;
    :  !EZ1/SP1 2.Setzhub nach Fraesen ;
    :  IF (F[335] AND F[78]),JMP LBL[55] ;
    :  !EZ1/SP1 Kurzschluss schweissen ;
    :  IF (F[335] AND !F[78]),JMP LBL[16] ;
    :  !EZ1/SP1 Kurzschluss schweissen ;
    :  IF (!F[335]),JMP LBL[16] ;
    :   ;
    :  !************************** ;
    :  !*       Schritt 16       * ;
    :  !*      STAT EZ1/SP1      * ;
    :  !* Kurzschlussschweissung * ;
    :  !************************** ;
    :   ;
    :  LBL[16] ;
    :  R[41]=16    ;
    :  !RSK gestartet ;
    :  F[321]=(OFF) ;
    :  DO[145]=(ON) ;
    :  !EZ1/SK1 Prog. ;
    :  IF (F[78] AND !F[301]),GO[1]=(41) ;
    :  IF (F[78] AND !F[301]),GO[3]=(41) ;
    :  IF (F[79] OR F[301]),GO[1]=(51) ;
    :  IF (F[79] OR F[301]),GO[3]=(51) ;
    :  WAIT    .10(sec) ;
    :  DO[717]=(OFF) ;
    :  DO[718]=(OFF) ;
    :  DO[785]=(OFF) ;
    :  DO[514]=(OFF) ;
    :  F[80]=(OFF) ;
    :  F[306]=(OFF) ;
    :  DO[18181]=(ON) ;
    :  WAIT (DI[705] AND DI[713] AND DI[714] AND (!DI[784] OR (DI[769] AND DI[784])))    ;
    :  DO[18181]=(OFF) ;
    :  F[346]=(OFF) ;
    :  DO[18181]=(ON) ;
    :  WAIT ((!DI[785] AND DI[792] AND DI[802] AND !F[80]) OR (!DI[792] AND DI[802] AND DI[145]))    ;
    :  DO[18181]=(OFF) ;
    :  !EZ1/SP1 schliessen ;
    :  DO[718]=(ON) ;
    :  TIMER[9]=((-4)) ;
    :  !EZ1/SP1 Kraft erreicht ;
    :  WAIT ((DI[718] AND !DI[772] AND !DI[780]) OR DI[774] OR DI[775] OR (TIMER[9]>=0))    ;
    :  DO[718]=(DI[718] AND !DI[774] AND !DI[775]) ;
    :  DO[717]=(!DO[718]) ;
    :  !Schweissen START ;
    :  DO[785]=(DI[718] AND !DI[774] AND !DI[775]) ;
    :  !EZ1/SP1 Fehler Ausgleich ;
    :  F[302]=(DI[718] AND DI[719]) ;
    :  !EZ1/SP1 Fehler SZ ;
    :  F[300]=(DI[774] OR DI[775]) ;
    :  !SK1 FK ;
    :  TIMER[9]=((-1)) ;
    :  WAIT ((F[80] AND DO[785]) OR ((DI[804] OR DI[805]) AND (DI[785] AND DO[785])) OR (DI[771] AND DI[784]) OR !DO[785] OR (TIMER[9]>=0))    ;
    :  F[297]=(F[80] OR (DI[804] AND !DI[806] AND !DI[775] AND DI[785])) ;
    :  !Fehler SK1 ;
    :  F[301]=(!F[297] AND !F[298] AND DO[785]) ;
    :  DO[785]=(OFF) ;
    :  DO[718]=(OFF) ;
    :  DO[18181]=(ON) ;
    :  F[749]=(!F[297] AND !F[748]) ;
    :  F[748]=(!F[297]) ;
    :  WAIT (F[297] OR DI[26] OR DI[27] OR (F[749] AND F[731]))    ;
    :  DO[910]=(OFF) ;
    :  WAIT (!DI[26] AND !DI[27])    ;
    :  DO[18181]=(OFF) ;
    :  !EZ1/SP1 oeffnen ;
    :  DO[717]=(!DI[717]) ;
    :  TIMER[9]=((-4)) ;
    :  WAIT (DI[717] OR (TIMER[9]>=0))    ;
    :  F[303]=((TIMER[9]>=0)) ;
    :  DO[18181]=(F[303]) ;
    :  WAIT (DI[717])    ;
    :  DO[18181]=(OFF) ;
    :  F[303]=(OFF) ;
    :  DO[717]=(OFF) ;
    :  DO[145]=(OFF) ;
    :  R[42]=16    ;
    :  JMP LBL[17] ;
    :   ;
    :  !************************** ;
    :  !*       Schritt 17       * ;
    :  !*      STAT EZ1/SP1      * ;
    :  !************************** ;
    :   ;
    :  LBL[17] ;
    :  R[41]=17    ;
    :  !RSK gestartet ;
    :  F[321]=(OFF) ;
    :  !Sprung zurueck bei Fehler ;
    :  IF (!F[297] AND !DI[777]),JMP LBL[9] ;
    :  !STAT EZ1/SP1 FK Fraesen ;
    :  F[93]=(!F[329]) ;
    :  DO[116]=(OFF) ;
    :  DO[130]=(OFF) ;
    :  R[42]=17    ;
    :  JMP LBL[1] ;
    :   ;
    :   ;
    :  !************************ ;
    :  !************************ ;
    :  !* Fraesen STAT EZ2/SP2 * ;
    :  !************************ ;
    :  !************************ ;
    :   ;
    :   ;
    :  !****************************** ;
    :  !*        Schritt 18          * ;
    :  !*     STAT EZ2/SP2 KS2       * ;
    :  !* KS2 in Arbeitsst.schwenken * ;
    :  !****************************** ;
    :   ;
    :  LBL[18] ;
    :  R[41]=18    ;
    :  !RSK gestartet ;
    :  F[321]=(OFF) ;
    :  GO[4]=(31) ;
    :  IF (F[285]),GO[3]=(35) ;
    :  IF (!F[285]),GO[6]=(31) ;
    :  WAIT    .10(sec) ;
    :  DO[918]=(F[138]) ;
    :  DO[919]=(F[139]) ;
    :  DO[116]=(ON) ;
    :  DO[162]=(ON) ;
    :  DO[878]=(OFF) ;
    :  DO[877]=(!DI[877]) ;
    :  DO[18181]=(ON) ;
    :  WAIT (DI[877])    ;
    :  DO[18181]=(OFF) ;
    :  DO[877]=(OFF) ;
    :  !Ueberwachungszeit Grundstellung ;
    :  TIMER[8]=((-4)) ;
    :  WAIT ((!DI[1004] AND DI[1002] AND DI[1005] AND !DI[1003]) OR (TIMER[8]>=0))    ;
    :  F[323]=((TIMER[8]>=0)) ;
    :  DO[18181]=((TIMER[8]>=0)) ;
    :  WAIT (!DI[1004] AND DI[1002] AND DI[1005] AND !DI[1003])    ;
    :  DO[18181]=(OFF) ;
    :  F[323]=(OFF) ;
    :  TIMER[8]=((-4)) ;
    :  DO[995]=(F[564]) ;
    :  WAIT ((DI[995] AND F[564]) OR (!DI[995] AND !F[564]) OR (TIMER[8]>=0))    ;
    :  F[323]=((TIMER[8]>=0)) ;
    :  DO[18181]=((TIMER[8]>=0)) ;
    :  WAIT ((DI[995] AND F[564]) OR (!DI[995] AND !F[564]))    ;
    :  DO[18181]=(OFF) ;
    :  F[323]=(OFF) ;
    :  !Ueberwachungszeit KS2 Schwenken ;
    :  TIMER[8]=((-6)) ;
    :  DO[3973]=(ON) ;
    :  DO[18181]=(ON) ;
    :  WAIT (DI[1001])    ;
    :  DO[18181]=(OFF) ;
    :  WAIT ((DI[1004] AND !DI[1002] AND !DI[1005] AND DI[1003]) OR (TIMER[8]>=0))    ;
    :  F[324]=((TIMER[8]>=0)) ;
    :  DO[3973]=(OFF) ;
    :  DO[18181]=((TIMER[8]>=0)) ;
    :  WAIT ((DI[1004] AND !DI[1002] AND !DI[1005] AND DI[1003]) OR DI[26])    ;
    :  DO[18181]=(OFF) ;
    :  F[324]=(OFF) ;
    :  !Sprung zurueck bei KS2 Fehler ;
    :  IF (TIMER[8]>=0),JMP LBL[18] ;
    :  DO[995]=(OFF) ;
    :  TIMER[11]=((R[24])) ;
    :  WAIT ((TIMER[11]>=0) OR !F[564])    ;
    :  TIMER[11]=STOP ;
    :  DO[18181]=(ON) ;
    :  WAIT ((F[148] AND F[138]) OR (F[148] AND F[139]))    ;
    :  DO[18181]=(OFF) ;
    :  !Anwahl Startfraesen ;
    :  IF (!DI[1002] AND DI[1003] AND F[148] AND F[138] AND !F[301]),R[41]=19 ;
    :  !Anwahl Normalfraesen ;
    :  IF (!DI[1002] AND DI[1003] AND F[148] AND (F[139] OR F[301])),R[41]=21 ;
    :  R[42]=18    ;
    :  JMP LBL[R[41]] ;
    :   ;
    :  !************************** ;
    :  !*      Schritt 19        * ;
    :  !* STAT EZ2/SP2 SF Teil 1 * ;
    :  !************************** ;
    :   ;
    :  LBL[19] ;
    :  R[41]=19    ;
    :  !RSK gestartet ;
    :  F[321]=(OFF) ;
    :  F[329]=(OFF) ;
    :  F[325]=(OFF) ;
    :  DO[878]=(OFF) ;
    :  DO[877]=(!DI[877]) ;
    :  DO[18181]=(ON) ;
    :  WAIT (DI[877])    ;
    :  DO[18181]=(OFF) ;
    :  DO[994]=(ON) ;
    :  DO[877]=(OFF) ;
    :  !Warte Fraeser laeuft ;
    :  TIMER[7]=((-3)) ;
    :  WAIT (!DI[994] OR (TIMER[7]>=0))    ;
    :  WAIT (DI[994] OR (TIMER[7]>=0))    ;
    :  F[322]=((TIMER[7]>=0)) ;
    :  DO[18181]=(ON) ;
    :  WAIT (!DI[994])    ;
    :  WAIT (DI[994])    ;
    :  DO[18181]=(OFF) ;
    :  F[322]=(OFF) ;
    :  !EZ2/SP2 schliessen ;
    :  DO[878]=(ON) ;
    :  !Fraeser ausblasen AUS/EIN ;
    :  DO[1007]=(F[330]) ;
    :  TIMER[9]=((-4)) ;
    :  !EZ2/SP2 Kraft erreicht ;
    :  WAIT ((DI[878] AND !DI[932] AND !DI[940] AND !DI[934] AND !DI[935]) OR (TIMER[9]>=0))    ;
    :  F[325]=((TIMER[9]>=0)) ;
    :  DO[18181]=(ON) ;
    :  DO[878]=((TIMER[9]<0)) ;
    :  DO[994]=((TIMER[9]<0)) ;
    :  WAIT ((DI[878] AND !DI[932] AND !DI[940] AND !DI[934] AND !DI[935]) OR DI[26] OR DI[27])    ;
    :  DO[18181]=(OFF) ;
    :  F[325]=(OFF) ;
    :  !EZ2/SP2 Fehler Kraftaufbau ;
    :  IF (F[325]),JMP LBL[1901] ;
    :  TIMER[9]=((-5)) ;
    :  LBL[1900] ;
    :  WAIT (!DI[994] OR F[325] OR (TIMER[9]>=0))    ;
    :  WAIT (DI[994] OR F[325] OR (TIMER[9]>=0))    ;
    :  R[1]=(R[1]+1) ;
    :  F[329]=((TIMER[9]>=0)) ;
    :  !Fraeszeit ueberschritten ;
    :  IF (F[329]),JMP LBL[1901] ;
    :  !Umdrehungen Vergleichen ;
    :  IF (R[1]<R[5]),JMP LBL[1900] ;
    :  F[150]=(ON) ;
    :  LBL[1901] ;
    :  DO[994]=((TIMER[9]<0)) ;
    :  !Fraeser ausblasen EIN ;
    :  DO[1007]=(F[330] OR (TIMER[9]<0)) ;
    :  DO[878]=(OFF) ;
    :  !EZ2/SP2 oeffnen ;
    :  DO[877]=(!DI[877]) ;
    :  DO[18181]=(F[329]) ;
    :  WAIT (!F[329] OR DI[26] OR DI[27])    ;
    :  DO[18181]=(OFF) ;
    :  DO[18181]=(ON) ;
    :  WAIT (DI[877])    ;
    :  DO[18181]=(OFF) ;
    :  DO[877]=(OFF) ;
    :  !Umdrehungen ruecksetzen ;
    :  R[1]=0    ;
    :  R[42]=19    ;
    :  IF (F[329] OR F[325]),JMP LBL[19] ;
    :  JMP LBL[20] ;
    :   ;
    :  !************************** ;
    :  !*       Schritt 20       * ;
    :  !* STAT EZ2/SP2 SF Teil 2 * ;
    :  !************************** ;
    :   ;
    :  LBL[20] ;
    :  R[41]=20    ;
    :  !RSK gestartet ;
    :  F[321]=(OFF) ;
    :  F[329]=(OFF) ;
    :  F[325]=(OFF) ;
    :  DO[878]=(OFF) ;
    :  DO[877]=(!DI[877]) ;
    :  DO[18181]=(ON) ;
    :  WAIT (DI[877])    ;
    :  DO[18181]=(OFF) ;
    :  DO[994]=(ON) ;
    :  DO[877]=(OFF) ;
    :  !Zange zu... ;
    :  DO[878]=(ON) ;
    :  !Fraeser ausblasen AUS/EIN ;
    :  DO[1007]=(F[330]) ;
    :  TIMER[9]=((-4)) ;
    :  !EZ2/SP2 Kraft erreicht ;
    :  WAIT ((DI[878] AND !DI[932] AND !DI[940] AND !DI[934] AND !DI[935]) OR (TIMER[9]>=0))    ;
    :  F[325]=((TIMER[9]>=0)) ;
    :  DO[18181]=(ON) ;
    :  DO[878]=((TIMER[9]<0)) ;
    :  DO[994]=((TIMER[9]<0)) ;
    :  WAIT ((DI[878] AND !DI[932] AND !DI[940] AND !DI[934] AND !DI[935]) OR DI[26] OR DI[27])    ;
    :  DO[18181]=(OFF) ;
    :  !EZ2/SP2 Fehler Kraftaufbau ;
    :  IF (F[325]),JMP LBL[2001] ;
    :  TIMER[9]=((-5)) ;
    :  LBL[2000] ;
    :  WAIT (!DI[994] OR F[325] OR (TIMER[9]>=0))    ;
    :  WAIT (DI[994] OR F[325] OR (TIMER[9]>=0))    ;
    :  R[1]=(R[1]+1) ;
    :  F[329]=((TIMER[9]>=0)) ;
    :  !Fraeszeit ueberschritten ;
    :  IF (F[329]),JMP LBL[2001] ;
    :  !Umdrehungen Vergleichen ;
    :  IF (R[1]<R[6]),JMP LBL[2000] ;
    :  F[152]=(ON) ;
    :  LBL[2001] ;
    :  DO[994]=((TIMER[9]<0)) ;
    :  !Fraeser ausblasen EIN ;
    :  DO[1007]=PULSE,4.0sec ;
    :  DO[878]=(OFF) ;
    :  !EZ2/SP2 oeffnen ;
    :  DO[877]=(!DI[877]) ;
    :  DO[18181]=(F[329]) ;
    :  WAIT (!F[329] OR DI[26] OR DI[27])    ;
    :  DO[18181]=(OFF) ;
    :  DO[18181]=(ON) ;
    :  WAIT (DI[877])    ;
    :  DO[18181]=(OFF) ;
    :  DO[877]=(OFF) ;
    :  !Umdrehungen ruecksetzen ;
    :  R[1]=0    ;
    :  R[42]=20    ;
    :  IF (F[329] OR F[325]),JMP LBL[20] ;
    :  JMP LBL[22] ;
    :   ;
    :  !********************* ;
    :  !*     Schritt 21    * ;
    :  !*   STAT EZ2/SP2 NF * ;
    :  !********************* ;
    :   ;
    :  LBL[21] ;
    :  R[41]=21    ;
    :  !RSK gestartet ;
    :  F[321]=(OFF) ;
    :  F[329]=(OFF) ;
    :  F[325]=(OFF) ;
    :  !Zähler wegspeichern für 2ten Hub ;
    :  R[45]=R[7]    ;
    :  IF (F[154] AND F[732]),R[7]=R[44] ;
    :  DO[878]=(OFF) ;
    :  DO[877]=(!DI[877]) ;
    :  DO[18181]=(ON) ;
    :  WAIT (DI[877])    ;
    :  DO[18181]=(OFF) ;
    :  DO[994]=(ON) ;
    :  DO[877]=(OFF) ;
    :  !EZ2/SP2 schliessen ;
    :  DO[878]=(ON) ;
    :  !Fraeser ausblasen AUS ;
    :  DO[1007]=(F[330]) ;
    :  TIMER[9]=((-4)) ;
    :  !EZ2/SP2 Kraft erreicht ;
    :  WAIT ((DI[878] AND !DI[932] AND !DI[940] AND !DI[934] AND !DI[935]) OR (TIMER[9]>=0))    ;
    :  F[325]=((TIMER[9]>=0)) ;
    :  DO[18181]=(ON) ;
    :  DO[878]=((TIMER[9]<0)) ;
    :  DO[994]=((TIMER[9]<0)) ;
    :  WAIT ((DI[878] AND !DI[932] AND !DI[940] AND !DI[934] AND !DI[935]) OR DI[26] OR DI[27])    ;
    :  DO[18181]=(OFF) ;
    :  !EZ2/SP2 Fehler Kraftaufbau ;
    :  IF (F[325]),JMP LBL[2101] ;
    :  TIMER[9]=((-5)) ;
    :  LBL[2100] ;
    :  WAIT (!DI[994] OR F[325] OR (TIMER[9]>=0))    ;
    :  WAIT (DI[994] OR F[325] OR (TIMER[9]>=0))    ;
    :  R[1]=(R[1]+1) ;
    :  F[329]=((TIMER[9]>=0)) ;
    :  !Fraeszeit ueberschritten ;
    :  IF (F[329]),JMP LBL[2101] ;
    :  !Umdrehungen Vergleichen ;
    :  IF (R[1]<R[7]),JMP LBL[2100] ;
    :  !EZ2/SP2 2 Huebe bei NF ;
    :  IF (!F[164]),JMP LBL[2101] ;
    :  IF (F[154]),F[152]=(ON) ;
    :  F[154]=(ON) ;
    :  LBL[2101] ;
    :  DO[878]=(OFF) ;
    :  DO[994]=((TIMER[9]<0)) ;
    :  !Fraeser ausblasen EIN ;
    :  DO[1007]=PULSE,4.0sec ;
    :  !EZ2/SP2 oeffnen ;
    :  DO[877]=(!DI[877]) ;
    :  DO[18181]=(F[329]) ;
    :  WAIT (!F[329] OR DI[26] OR DI[27])    ;
    :  DO[18181]=(OFF) ;
    :  DO[18181]=(ON) ;
    :  WAIT (DI[877])    ;
    :  DO[18181]=(OFF) ;
    :  DO[877]=(OFF) ;
    :  !Umdrehungen ruecksetzen ;
    :  R[1]=0    ;
    :  R[42]=21    ;
    :  !Zähler umschreiben für 2ten Hub ;
    :  IF (F[154] AND F[732]),GO[3]=36 ;
    :  IF (F[152] AND F[732]),R[7]=R[45] ;
    :  IF (F[329] OR F[325] OR (!F[152] AND F[164])),JMP LBL[21] ;
    :  F[154]=(ON) ;
    :  JMP LBL[22] ;
    :   ;
    :  !*************************** ;
    :  !*        Schritt 22       * ;
    :  !* STAT EZ2/SP2 i.O/n.i.O. * ;
    :  !*************************** ;
    :   ;
    :  LBL[22] ;
    :  R[41]=22    ;
    :  !Fraesueberwachung starten ;
    :  TIMER[7]=((-5)) ;
    :  WAIT ((F[138] OR F[139]) AND (F[154] OR (F[150] AND F[152])) OR (TIMER[7]>=0))    ;
    :  F[329]=((TIMER[7]>=0)) ;
    :  IF (!F[329]),R[41]=23 ;
    :  IF (F[329]),R[41]=21 ;
    :  !KF1 U-Merker ruecksetzen ;
    :  F[150]=(OFF) ;
    :  F[152]=(OFF) ;
    :  F[154]=(OFF) ;
    :  R[42]=22    ;
    :  JMP LBL[R[41]] ;
    :   ;
    :  !*************************** ;
    :  !*       Schritt 23        * ;
    :  !*      STAT EZ2/SP2       * ;
    :  !* KS2 in Ruhest.schwenken * ;
    :  !*************************** ;
    :   ;
    :  LBL[23] ;
    :  R[41]=23    ;
    :  !RSK gestartet ;
    :  F[321]=(OFF) ;
    :  DO[878]=(OFF) ;
    :  DO[877]=(!DI[877]) ;
    :  DO[18181]=(ON) ;
    :  WAIT (DI[877])    ;
    :  DO[18181]=(OFF) ;
    :  DO[877]=(OFF) ;
    :  TIMER[8]=((-4)) ;
    :  WAIT ((DI[1004] AND !DI[1002] AND !DI[1005] AND DI[1003]) OR (TIMER[8]>=0))    ;
    :  F[324]=((TIMER[8]>=0)) ;
    :  DO[18181]=((TIMER[8]>=0)) ;
    :  WAIT (DI[1004] AND !DI[1002] AND !DI[1005] AND DI[1003])    ;
    :  DO[18181]=(OFF) ;
    :  F[324]=(OFF) ;
    :  TIMER[8]=((-4)) ;
    :  DO[995]=(F[564]) ;
    :  WAIT ((DI[995] AND F[564]) OR (!DI[995] AND !F[564]) OR (TIMER[8]>=0))    ;
    :  F[323]=((TIMER[8]>=0)) ;
    :  DO[18181]=((TIMER[8]>=0)) ;
    :  WAIT ((DI[995] AND F[564]) OR (!DI[995] AND !F[564]))    ;
    :  DO[18181]=(OFF) ;
    :  F[323]=(OFF) ;
    :  !Ueberwachungszeit KS2 Schwenken ;
    :  TIMER[8]=((-4)) ;
    :  DO[3970]=(ON) ;
    :  WAIT (DI[1001] OR (TIMER[8]>=0))    ;
    :  DO[18181]=((TIMER[8]>=0)) ;
    :  WAIT (DI[1001])    ;
    :  TIMER[8]=((-6)) ;
    :  DO[18181]=(OFF) ;
    :  WAIT ((!DI[1004] AND DI[1002] AND DI[1005] AND !DI[1003]) OR (TIMER[8]>=0))    ;
    :  F[323]=((TIMER[8]>=0)) ;
    :  DO[3970]=(OFF) ;
    :  DO[18181]=((TIMER[8]>=0)) ;
    :  WAIT ((!DI[1004] AND DI[1002] AND DI[1005] AND !DI[1003]) OR DI[26])    ;
    :  DO[18181]=(OFF) ;
    :  F[323]=(OFF) ;
    :  DO[995]=(OFF) ;
    :  DO[994]=(OFF) ;
    :  !Sprung zurueck bei KS2 Fehler ;
    :  IF (TIMER[8]>=0),JMP LBL[23] ;
    :  R[42]=23    ;
    :  JMP LBL[24] ;
    :   ;
    :  !*********************** ;
    :  !*     Schritt 24      * ;
    :  !*    STAT EZ2/SP2     * ;
    :  !* Messen nach Fraesen * ;
    :  !*********************** ;
    :   ;
    :  LBL[24] ;
    :  R[41]=24    ;
    :  !RSK gestartet ;
    :  F[321]=(OFF) ;
    :  IF (!F[285]),JMP LBL[2400] ;
    :  IF (F[285]),JMP LBL[2401] ;
    :  LBL[2400] ;
    :  GO[6]=1 ;
    :  WAIT    .10(sec) ;
    :  DO[946]=(ON) ;
    :  !STAT EZ2/SP2 FK Fraesen ;
    :  DO[18181]=(ON) ;
    :  WAIT (!DI[946] AND DI[947] AND !DI[948])    ;
    :  DO[18181]=(OFF) ;
    :  DO[946]=(OFF) ;
    :  JMP LBL[2402] ;
    :  LBL[2401] ;
    :  IF (!F[285]),GO[3]=(1) ;
    :  IF (F[285]),GO[3]=(5) ;
    :  WAIT    .10(sec) ;
    :  DO[786]=(ON) ;
    :  !STAT EZ2/SP2 FK Fraesen ;
    :  DO[18181]=(ON) ;
    :  WAIT (!DI[786] AND DI[787] AND !DI[788])    ;
    :  DO[18181]=(OFF) ;
    :  DO[786]=(OFF) ;
    :  LBL[2402] ;
    :  GO[4]=(31) ;
    :  IF (F[285]),GO[3]=(35) ;
    :  IF (!F[285]),GO[6]=(31) ;
    :  WAIT    .10(sec) ;
    :  DO[917]=(ON) ;
    :  TIMER[9]=((-8)) ;
    :  WAIT (DI[917] OR (TIMER[9]>=0))    ;
    :  F[326]=((TIMER[9]>=0)) ;
    :  DO[18181]=(F[326]) ;
    :  WAIT (DI[917] OR DI[26] OR DI[27])    ;
    :  DO[18181]=(OFF) ;
    :  F[326]=(OFF) ;
    :  F[143]=(DI[936] OR DI[937]) ;
    :  DO[917]=(OFF) ;
    :  F[144]=(DI[896] OR (DI[895] AND DI[894] AND DI[893])) ;
    :  TIMER[7]=((-2)) ;
    :  WAIT ((!F[144] AND !F[143]) OR (TIMER[7]>=0))    ;
    :  F[329]=((TIMER[7]>=0)) ;
    :  DO[18181]=(F[329]) ;
    :  WAIT ((!F[144] AND !F[143]) OR DI[26] OR DI[27])    ;
    :  DO[18181]=(OFF) ;
    :  F[329]=(OFF) ;
    :  F[298]=(F[144] OR F[143]) ;
    :  DO[877]=(!DI[877]) ;
    :  DO[18181]=(ON) ;
    :  WAIT ((DI[877] AND !DI[944]) OR (DI[877] AND F[298]))    ;
    :  DO[18181]=(OFF) ;
    :  DO[877]=(OFF) ;
    :  R[42]=24    ;
    :  !EZ2/SP2 wiederh. bei Messfehler ;
    :  IF (F[298]),JMP LBL[18] ;
    :  DO[918]=(OFF) ;
    :  DO[919]=(OFF) ;
    :  !KS nicht bei K-Verschleiss ;
    :  IF (DI[937]),JMP LBL[26] ;
    :  !EZ2/SP2 2.Setzhub nach Fraesen ;
    :  IF (F[335] AND F[138]),JMP LBL[56] ;
    :  !EZ2/SP2 Kurzschluss schweissen ;
    :  IF (F[335] AND !F[138]),JMP LBL[25] ;
    :  !EZ2/SP2 Kurzschluss schweissen ;
    :  IF (!F[335]),JMP LBL[25] ;
    :   ;
    :  !************************** ;
    :  !*       Schritt 25       * ;
    :  !*      STAT EZ2/SP2      * ;
    :  !* Kurzschlussschweissung * ;
    :  !************************** ;
    :   ;
    :  LBL[25] ;
    :  R[41]=25    ;
    :  !RSK gestartet ;
    :  F[321]=(OFF) ;
    :  DO[145]=(F[285]) ;
    :  DO[177]=(!F[285]) ;
    :  !EZ2/SP2 SK1/SK2 Prog. ;
    :  IF (F[285] AND F[138] AND !F[301]),GO[3]=(45) ;
    :  IF (!F[285] AND F[138] AND !F[301]),GO[4]=(41) ;
    :  IF (!F[285] AND F[138] AND !F[301]),GO[6]=(41) ;
    :  IF ((F[285] AND F[139]) OR (F[285] AND F[301])),GO[3]=(55) ;
    :  IF ((!F[285] AND F[139]) OR (!F[285] AND F[301])),GO[4]=(51) ;
    :  IF ((!F[285] AND F[139]) OR (!F[285] AND F[301])),GO[6]=(51) ;
    :  WAIT    .10(sec) ;
    :  DO[877]=(OFF) ;
    :  DO[878]=(OFF) ;
    :  DO[945]=(OFF) ;
    :  DO[785]=(!F[285] AND DO[785]) ;
    :  DO[514]=(ON) ;
    :  F[140]=(OFF) ;
    :  F[80]=(OFF) ;
    :  F[142]=(!F[285]) ;
    :  F[306]=(OFF) ;
    :  F[303]=(!DI[929] AND DI[944]) ;
    :  DO[18181]=(ON) ;
    :  WAIT (DI[865] AND DI[873] AND DI[874] AND (!DI[944] OR (DI[929] AND DI[944])))    ;
    :  F[303]=(OFF) ;
    :  WAIT ((!DI[945] AND DI[952] AND DI[962] AND !F[140]) OR (!DI[952] AND DI[962] AND !DI[913]) OR F[285])    ;
    :  WAIT ((!DI[785] AND DI[792] AND DI[802] AND !F[80]) OR (!DI[792] AND DI[802] AND !DI[913]) OR !F[285])    ;
    :  DO[18181]=(OFF) ;
    :  !EZ2/SP2 schliessen ;
    :  DO[878]=(ON) ;
    :  TIMER[9]=((-4)) ;
    :  WAIT ((DI[878] AND !DI[932] AND !DI[940]) OR DI[934] OR DI[935] OR (TIMER[9]>=0))    ;
    :  DO[878]=(DI[878] AND !DI[934] AND !DI[935]) ;
    :  DO[877]=(!DO[878]) ;
    :  !Schweissen START ;
    :  DO[945]=(DI[878] AND !DI[934] AND !DI[935] AND !F[285]) ;
    :  DO[785]=((DI[878] AND !DI[934] AND !DI[935] AND F[285]) OR (!F[285] AND DO[785])) ;
    :  !EZ2/SP2 Fehler Ausgleich ;
    :  F[302]=(DI[878] AND DI[879]) ;
    :  !EZ2/SP2 Fehler SZ ;
    :  F[300]=(DI[934] OR DI[935]) ;
    :  !SK1/SK2 FK ;
    :  TIMER[9]=((-10)) ;
    :  WAIT ((F[140] AND DO[945]) OR ((DI[964] OR DI[965]) AND (DI[945] AND DO[945])) OR (DI[931] AND DI[944]) OR (!DO[945] AND F[285]) OR (TIMER[9]>=0))    ;
    :  WAIT ((F[80] AND DO[785]) OR ((DI[804] OR DI[805]) AND (DI[785] AND DO[785])) OR (DI[931] AND DI[944]) OR (!DO[785] AND !F[285]) OR (TIMER[9]>=0))    ;
    :  F[297]=(F[140] OR (!DI[935] AND DI[945] AND DI[964] AND !DI[966]) OR F[80] OR (!DI[935] AND DI[785] AND DI[804] AND !DI[806])) ;
    :  !Fehler SK1/SK2 ;
    :  F[301]=(!F[297] AND !F[298] AND (DO[785] OR DO[945])) ;
    :  DO[945]=(OFF) ;
    :  DO[878]=(OFF) ;
    :  DO[785]=((F[285] AND !DI[785]) OR (!F[285] AND DO[785])) ;
    :  F[327]=(!F[297]) ;
    :  DO[18181]=(F[327]) ;
    :  F[749]=(!F[297] AND !F[748]) ;
    :  F[748]=(!F[297]) ;
    :  WAIT (F[297] OR DI[26] OR DI[27] OR (F[749] AND F[731]))    ;
    :  F[327]=(OFF) ;
    :  WAIT (!DI[26] AND !DI[27])    ;
    :  DO[18181]=(OFF) ;
    :  !EZ2/SP2 oeffnen ;
    :  DO[877]=(!DI[877]) ;
    :  TIMER[9]=((-4)) ;
    :  WAIT (DI[877] OR (TIMER[9]>=0))    ;
    :  F[303]=((TIMER[9]>=0)) ;
    :  DO[18181]=(F[303]) ;
    :  WAIT (DI[877])    ;
    :  DO[18181]=(OFF) ;
    :  F[303]=(OFF) ;
    :  DO[877]=(OFF) ;
    :  DO[145]=(OFF) ;
    :  DO[177]=(OFF) ;
    :  R[42]=25    ;
    :  JMP LBL[26] ;
    :   ;
    :  !****************************** ;
    :  !*         Schritt 26         * ;
    :  !*       STAT EZ2/SP2 FK      * ;
    :  !****************************** ;
    :   ;
    :  LBL[26] ;
    :  R[41]=26    ;
    :  !RSK gestartet ;
    :  F[321]=(OFF) ;
    :  !Sprung zurueck bei Fehler ;
    :  IF (!F[297] AND !DI[937]),JMP LBL[18] ;
    :  !STAT EZ2/SP2 FK Fraesen ;
    :  F[149]=(!F[329]) ;
    :  DO[116]=(OFF) ;
    :  DO[162]=(OFF) ;
    :  R[42]=26    ;
    :  JMP LBL[1] ;
    :   ;
    :   ;
    :  !************************ ;
    :  !************************ ;
    :  !* Fraesen STAT EZ3/SP3 * ;
    :  !************************ ;
    :  !************************ ;
    :   ;
    :   ;
    :  !******************************* ;
    :  !*        Schritt 27           * ;
    :  !*       STAT EZ3/SP3          * ;
    :  !* KS3 in Arbeitsst. schwenken * ;
    :  !******************************* ;
    :   ;
    :  LBL[27] ;
    :  R[41]=27    ;
    :  !RSK gestartet ;
    :  F[321]=(OFF) ;
    :  GO[7]=(31) ;
    :  GO[9]=(31) ;
    :  WAIT    .10(sec) ;
    :  DO[1078]=(F[174]) ;
    :  DO[1079]=(F[175]) ;
    :  DO[116]=(ON) ;
    :  DO[194]=(ON) ;
    :  DO[1038]=(OFF) ;
    :  DO[1037]=(!DI[1037]) ;
    :  DO[18181]=(ON) ;
    :  WAIT (DI[1037])    ;
    :  DO[18181]=(OFF) ;
    :  DO[1037]=(OFF) ;
    :  !Ueberwachungszeit Grundstellung ;
    :  TIMER[8]=((-4)) ;
    :  WAIT ((DI[1162] AND !DI[1163] AND !DI[1164] AND DI[1165]) OR (TIMER[8]>=0))    ;
    :  F[323]=((TIMER[8]>=0)) ;
    :  DO[18181]=((TIMER[8]>=0)) ;
    :  WAIT (DI[1162] AND !DI[1163] AND !DI[1164] AND DI[1165])    ;
    :  DO[18181]=(OFF) ;
    :  F[323]=(OFF) ;
    :  TIMER[8]=((-4)) ;
    :  DO[1155]=(F[564]) ;
    :  WAIT ((DI[1155] AND F[564]) OR (!DI[1155] AND !F[564]) OR (TIMER[8]>=0))    ;
    :  F[323]=((TIMER[8]>=0)) ;
    :  DO[18181]=((TIMER[8]>=0)) ;
    :  WAIT ((DI[1155] AND F[564]) OR (!DI[1155] AND !F[564]))    ;
    :  DO[18181]=(OFF) ;
    :  F[323]=(OFF) ;
    :  !Ueberwachungszeit KS3 Schwenken ;
    :  TIMER[8]=((-4)) ;
    :  DO[3974]=(ON) ;
    :  WAIT (DI[1161] OR (TIMER[8]>=0))    ;
    :  DO[18181]=((TIMER[8]>=0)) ;
    :  WAIT (DI[1161])    ;
    :  TIMER[8]=((-6)) ;
    :  DO[18181]=(OFF) ;
    :  WAIT ((!DI[1162] AND DI[1163] AND DI[1164] AND !DI[1165]) OR (TIMER[8]>=0))    ;
    :  F[324]=((TIMER[8]>=0)) ;
    :  DO[3974]=(OFF) ;
    :  DO[18181]=((TIMER[8]>=0)) ;
    :  WAIT ((!DI[1162] AND DI[1163] AND DI[1164] AND !DI[1165]) OR DI[26])    ;
    :  DO[18181]=(OFF) ;
    :  F[324]=(OFF) ;
    :  !Sprung zurueck bei KS3 Fehler ;
    :  IF (TIMER[8]>=0),JMP LBL[27] ;
    :  DO[1155]=(OFF) ;
    :  TIMER[11]=((R[24])) ;
    :  WAIT ((TIMER[11]>=0) OR !F[564])    ;
    :  TIMER[11]=STOP ;
    :  DO[18181]=(ON) ;
    :  WAIT ((F[184] AND F[174]) OR (F[184] AND F[175]))    ;
    :  DO[18181]=(OFF) ;
    :  !Anwahl Startfraesen ;
    :  IF (!DI[1162] AND DI[1163] AND F[184] AND F[174] AND !F[301]),R[41]=28 ;
    :  !Anwahl Normalfraesen ;
    :  IF (!DI[1162] AND DI[1163] AND F[184] AND (F[175] OR F[301])),R[41]=30 ;
    :  R[42]=27    ;
    :  JMP LBL[R[41]] ;
    :   ;
    :  !************************** ;
    :  !*       Schritt 28       * ;
    :  !* STAT EZ3/SP3 SF Teil 1 * ;
    :  !************************** ;
    :   ;
    :  LBL[28] ;
    :  R[41]=28    ;
    :  !RSK gestartet ;
    :  F[321]=(OFF) ;
    :  F[329]=(OFF) ;
    :  F[325]=(OFF) ;
    :  DO[1038]=(OFF) ;
    :  DO[1037]=(!DI[1037]) ;
    :  DO[18181]=(ON) ;
    :  WAIT (DI[1037])    ;
    :  DO[1037]=(OFF) ;
    :  DO[18181]=(OFF) ;
    :  DO[1154]=(ON) ;
    :  !Warte Fraeser laeuft ;
    :  TIMER[7]=((-3)) ;
    :  WAIT (!DI[1154] OR (TIMER[7]>=0))    ;
    :  WAIT (DI[1154] OR (TIMER[7]>=0))    ;
    :  F[322]=((TIMER[7]>=0)) ;
    :  DO[18181]=(ON) ;
    :  WAIT (!DI[1154])    ;
    :  WAIT (DI[1154])    ;
    :  DO[18181]=(OFF) ;
    :  F[322]=(OFF) ;
    :  !EZ3/SP3 schliessen ;
    :  DO[1038]=(ON) ;
    :  !Fraeser ausblasen AUS/EIN ;
    :  DO[1167]=(F[330]) ;
    :  TIMER[9]=((-4)) ;
    :  !EZ3/SP3 Kraft erreicht ;
    :  WAIT ((DI[1038] AND !DI[1092] AND !DI[1100] AND !DI[1094] AND !DI[1095]) OR (TIMER[9]>=0))    ;
    :  F[325]=((TIMER[9]>=0)) ;
    :  DO[18181]=(ON) ;
    :  DO[1038]=((TIMER[9]<0)) ;
    :  DO[1154]=((TIMER[9]<0)) ;
    :  WAIT ((DI[1038] AND !DI[1092] AND !DI[1100] AND !DI[1094] AND !DI[1095]) OR DI[26] OR DI[27])    ;
    :  DO[18181]=(OFF) ;
    :  !EZ3/SP3 Fehler Kraftaufbau ;
    :  IF (F[325]),JMP LBL[2801] ;
    :  TIMER[9]=((-5)) ;
    :  LBL[2800] ;
    :  WAIT (!DI[1154] OR F[325] OR (TIMER[9]>=0))    ;
    :  WAIT (DI[1154] OR F[325] OR (TIMER[9]>=0))    ;
    :  R[1]=(R[1]+1) ;
    :  F[329]=((TIMER[9]>=0)) ;
    :  !Fraeszeit ueberschritten ;
    :  IF (F[329]),JMP LBL[2801] ;
    :  !Umdrehungen Vergleichen ;
    :  IF (R[1]<R[17]),JMP LBL[2800] ;
    :  F[186]=(ON) ;
    :  LBL[2801] ;
    :  DO[1154]=((TIMER[9]<0)) ;
    :  !Fraeser ausblasen EIN ;
    :  DO[1167]=(F[330] OR (TIMER[9]<0)) ;
    :  DO[1038]=(OFF) ;
    :  !EZ3/SP3 oeffnen ;
    :  DO[1037]=(!DI[1037]) ;
    :  DO[18181]=(F[329]) ;
    :  WAIT (!F[329] OR DI[26] OR DI[27])    ;
    :  DO[18181]=(OFF) ;
    :  DO[18181]=(ON) ;
    :  WAIT (DI[1037])    ;
    :  DO[18181]=(OFF) ;
    :  DO[1037]=(OFF) ;
    :  !Umdrehungen ruecksetzen ;
    :  R[1]=0    ;
    :  R[42]=28    ;
    :  IF (F[329] OR F[325]),JMP LBL[28] ;
    :  JMP LBL[29] ;
    :   ;
    :  !************************** ;
    :  !*      Schritt 29        * ;
    :  !* STAT EZ3/SP3 SF Teil 2 * ;
    :  !************************** ;
    :   ;
    :  LBL[29] ;
    :  R[41]=29    ;
    :  !RSK gestartet ;
    :  F[321]=(OFF) ;
    :  F[329]=(OFF) ;
    :  F[325]=(OFF) ;
    :  DO[1038]=(OFF) ;
    :  DO[1037]=(!DI[1037]) ;
    :  DO[18181]=(ON) ;
    :  WAIT (DI[1037])    ;
    :  DO[18181]=(OFF) ;
    :  DO[1154]=(ON) ;
    :  DO[1037]=(OFF) ;
    :  !EZ3/SP3 schliessen ;
    :  DO[1038]=(ON) ;
    :  !Fraeser ausblasen AUS/EIN ;
    :  DO[1167]=(F[330]) ;
    :  TIMER[9]=((-4)) ;
    :  !EZ3/SP3 Kraft erreicht ;
    :  WAIT ((DI[1038] AND !DI[1092] AND !DI[1100] AND !DI[1094] AND !DI[1095]) OR (TIMER[9]>=0))    ;
    :  F[325]=((TIMER[9]>=0)) ;
    :  DO[18181]=(ON) ;
    :  DO[1038]=((TIMER[9]<0)) ;
    :  DO[1154]=((TIMER[9]<0)) ;
    :  WAIT ((DI[1038] AND !DI[1092] AND !DI[1100] AND !DI[1094] AND !DI[1095]) OR DI[26] OR DI[27])    ;
    :  DO[18181]=(OFF) ;
    :  !EZ3/SP3 Fehler Kraftaufbau ;
    :  IF (F[325]),JMP LBL[2901] ;
    :  TIMER[9]=((-5)) ;
    :  LBL[2900] ;
    :  WAIT (!DI[1154] OR F[325] OR (TIMER[9]>=0))    ;
    :  WAIT (DI[1154] OR F[325] OR (TIMER[9]>=0))    ;
    :  R[1]=(R[1]+1) ;
    :  F[329]=((TIMER[9]>=0)) ;
    :  !Fraeszeit ueberschritten ;
    :  IF (F[329]),JMP LBL[2901] ;
    :  !Umdrehungen Vergleichen ;
    :  IF (R[1]<R[18]),JMP LBL[2900] ;
    :  F[188]=(ON) ;
    :  LBL[2901] ;
    :  DO[1154]=((TIMER[9]<0)) ;
    :  !Fraeser ausblasen EIN ;
    :  DO[1167]=PULSE,4.0sec ;
    :  DO[1038]=(OFF) ;
    :  !EZ3/SP3 oeffnen ;
    :  DO[1037]=(!DI[1037]) ;
    :  DO[18181]=(F[329]) ;
    :  WAIT (!F[329] OR DI[26] OR DI[27])    ;
    :  DO[18181]=(OFF) ;
    :  DO[18181]=(ON) ;
    :  WAIT (DI[1037])    ;
    :  DO[18181]=(OFF) ;
    :  DO[1037]=(OFF) ;
    :  !Umdrehungen ruecksetzen ;
    :  R[1]=0    ;
    :  R[42]=29    ;
    :  IF (F[329] OR F[325]),JMP LBL[29] ;
    :  JMP LBL[31] ;
    :   ;
    :  !******************* ;
    :  !*   Schritt 30    * ;
    :  !* STAT EZ3/SP3 NF * ;
    :  !******************* ;
    :   ;
    :  LBL[30] ;
    :  R[41]=30    ;
    :  !RSK gestartet ;
    :  F[321]=(OFF) ;
    :  F[329]=(OFF) ;
    :  F[325]=(OFF) ;
    :  !Zähler wegspeichern für 2ten Hub ;
    :  R[45]=R[19]    ;
    :  IF (F[190] AND F[732]),R[19]=R[38] ;
    :  DO[1038]=(OFF) ;
    :  DO[1037]=(!DI[1037]) ;
    :  DO[18181]=(ON) ;
    :  WAIT (DI[1037])    ;
    :  DO[18181]=(OFF) ;
    :  DO[1154]=(ON) ;
    :  DO[1037]=(OFF) ;
    :  !EZ3/SP3 schliessen ;
    :  DO[1038]=(ON) ;
    :  !Fraeser ausblasen AUS ;
    :  DO[1167]=(F[330]) ;
    :  TIMER[9]=((-4)) ;
    :  !EZ3/SP3 Kraft erreicht ;
    :  WAIT ((DI[1038] AND !DI[1092] AND !DI[1100] AND !DI[1094] AND !DI[1095]) OR (TIMER[9]>=0))    ;
    :  F[325]=((TIMER[9]>=0)) ;
    :  DO[18181]=(ON) ;
    :  DO[1038]=((TIMER[9]<0)) ;
    :  DO[1154]=((TIMER[9]<0)) ;
    :  WAIT ((DI[1038] AND !DI[1092] AND !DI[1100] AND !DI[1094] AND !DI[1095]) OR DI[26] OR DI[27])    ;
    :  DO[18181]=(OFF) ;
    :  !EZ3/SP3 Fehler Kraftaufbau ;
    :  IF (F[325]),JMP LBL[3001] ;
    :  TIMER[9]=((-5)) ;
    :  LBL[3000] ;
    :  WAIT (!DI[1154] OR F[325] OR (TIMER[9]>=0))    ;
    :  WAIT (DI[1154] OR F[325] OR (TIMER[9]>=0))    ;
    :  R[1]=(R[1]+1) ;
    :  F[329]=((TIMER[9]>=0)) ;
    :  !Fraeszeit ueberschritten ;
    :  IF (F[329]),JMP LBL[3001] ;
    :  !Umdrehungen Vergleichen ;
    :  IF (R[1]<R[19]),JMP LBL[3000] ;
    :  !EZ3/SP3 2 Huebe bei NF ;
    :  IF (!F[200]),JMP LBL[3001] ;
    :  IF (F[190]),F[188]=(ON) ;
    :  F[190]=(ON) ;
    :  LBL[3001] ;
    :  DO[1154]=((TIMER[9]<0)) ;
    :  !Fraeser ausblasen EIN ;
    :  DO[1167]=PULSE,4.0sec ;
    :  !EZ3/SP3 oeffnen ;
    :  DO[1038]=(OFF) ;
    :  DO[1037]=(!DI[1037]) ;
    :  DO[18181]=(F[329]) ;
    :  WAIT (!F[329] OR DI[26] OR DI[27])    ;
    :  DO[18181]=(OFF) ;
    :  DO[18181]=(ON) ;
    :  WAIT (DI[1037])    ;
    :  DO[18181]=(OFF) ;
    :  DO[1037]=(OFF) ;
    :  !Umdrehungen ruecksetzen ;
    :  R[1]=0    ;
    :  R[42]=30    ;
    :  IF (F[190] AND F[732]),GO[3]=36 ;
    :  IF (F[188] AND F[732]),R[19]=R[45] ;
    :  IF (F[329] OR F[325] OR (!F[188] AND F[200])),JMP LBL[30] ;
    :  F[190]=(ON) ;
    :  JMP LBL[31] ;
    :   ;
    :  !**************************** ;
    :  !*        Schritt 31        * ;
    :  !* STAT EZ3/SP3 i.O./n.i.O. * ;
    :  !**************************** ;
    :   ;
    :  LBL[31] ;
    :  R[41]=31    ;
    :  !Fraesueberwachung starten ;
    :  TIMER[7]=((-5)) ;
    :  WAIT ((F[174] OR F[175]) AND (F[190] OR (F[186] AND F[188])) OR (TIMER[7]>=0))    ;
    :  F[329]=((TIMER[7]>=0)) ;
    :  IF (!F[329]),R[41]=32 ;
    :  IF (F[329]),R[41]=30 ;
    :  !KF1 U-Merker ruecksetzen ;
    :  F[186]=(OFF) ;
    :  F[188]=(OFF) ;
    :  F[190]=(OFF) ;
    :  R[42]=31    ;
    :  JMP LBL[R[41]] ;
    :   ;
    :  !**************************** ;
    :  !*       Schritt 32         * ;
    :  !*      STAT EZ3/SP3        * ;
    :  !* KS3 in Ruhest. schwenken * ;
    :  !**************************** ;
    :   ;
    :  LBL[32] ;
    :  R[41]=32    ;
    :  !RSK gestartet ;
    :  F[321]=(OFF) ;
    :  DO[1038]=(OFF) ;
    :  DO[1037]=(!DI[1037]) ;
    :  DO[18181]=(ON) ;
    :  WAIT (DI[1037])    ;
    :  DO[18181]=(OFF) ;
    :  DO[1037]=(OFF) ;
    :  TIMER[8]=((-4)) ;
    :  WAIT ((DI[1164] AND !DI[1162] AND !DI[1165] AND DI[1163]) OR (TIMER[8]>=0))    ;
    :  F[324]=((TIMER[8]>=0)) ;
    :  DO[18181]=((TIMER[8]>=0)) ;
    :  WAIT (DI[1164] AND !DI[1162] AND !DI[1165] AND DI[1163])    ;
    :  DO[18181]=(OFF) ;
    :  F[324]=(OFF) ;
    :  TIMER[8]=((-4)) ;
    :  DO[1155]=(F[564]) ;
    :  WAIT ((DI[1155] AND F[564]) OR (!DI[1155] AND !F[564]) OR (TIMER[8]>=0))    ;
    :  F[323]=((TIMER[8]>=0)) ;
    :  DO[18181]=((TIMER[8]>=0)) ;
    :  WAIT ((DI[1155] AND F[564]) OR (!DI[1155] AND !F[564]))    ;
    :  DO[18181]=(OFF) ;
    :  F[323]=(OFF) ;
    :  !Ueberwachungszeit KS3 Schwenken ;
    :  TIMER[8]=((-4)) ;
    :  DO[3971]=(ON) ;
    :  WAIT (DI[1161] OR (TIMER[8]>=0))    ;
    :  DO[18181]=((TIMER[8]>=0)) ;
    :  WAIT (DI[1161])    ;
    :  TIMER[8]=((-6)) ;
    :  DO[18181]=(OFF) ;
    :  WAIT ((!DI[1164] AND DI[1162] AND DI[1165] AND !DI[1163]) OR (TIMER[8]>=0))    ;
    :  F[323]=((TIMER[8]>=0)) ;
    :  DO[3971]=(OFF) ;
    :  DO[18181]=((TIMER[8]>=0)) ;
    :  WAIT ((!DI[1164] AND DI[1162] AND DI[1165] AND !DI[1163]) OR DI[26])    ;
    :  DO[18181]=(OFF) ;
    :  F[323]=(OFF) ;
    :  DO[1154]=(OFF) ;
    :  DO[1155]=(OFF) ;
    :  !Sprung zurueck bei KS3 Fehler ;
    :  IF (TIMER[8]>=0),JMP LBL[32] ;
    :  R[42]=32    ;
    :  JMP LBL[33] ;
    :   ;
    :  !*********************** ;
    :  !*     Schritt 33      * ;
    :  !*    STAT EZ3/SP3     * ;
    :  !* Messen nach Fraesen * ;
    :  !*********************** ;
    :   ;
    :  LBL[33] ;
    :  R[41]=33    ;
    :  !RSK gestartet ;
    :  F[321]=(OFF) ;
    :  GO[9]=1 ;
    :  WAIT    .10(sec) ;
    :  DO[1106]=(ON) ;
    :  !STAT EZ3/SP3 FK Fraesen ;
    :  DO[18181]=(ON) ;
    :  WAIT (!DI[1106] AND DI[1107] AND !DI[1108])    ;
    :  DO[18181]=(OFF) ;
    :  DO[1106]=(OFF) ;
    :  GO[7]=(31) ;
    :  GO[9]=(31) ;
    :  WAIT    .10(sec) ;
    :  DO[1077]=(ON) ;
    :  TIMER[9]=((-8)) ;
    :  WAIT (DI[1077] OR (TIMER[9]>=0))    ;
    :  DO[326]=((TIMER[9]>=0)) ;
    :  DO[18181]=(ON) ;
    :  WAIT (DI[1077] OR DI[26] OR DI[27])    ;
    :  DO[18181]=(OFF) ;
    :  DO[326]=(OFF) ;
    :  F[179]=(DI[1096] OR DI[1097]) ;
    :  DO[1077]=(OFF) ;
    :  F[180]=(DI[1056] OR (DI[1055] AND DI[1054] AND DI[1053])) ;
    :  TIMER[7]=((-2)) ;
    :  WAIT ((!F[180] AND !F[179]) OR (TIMER[7]>=0))    ;
    :  F[329]=((TIMER[7]>=0)) ;
    :  DO[18181]=(F[329]) ;
    :  WAIT ((!F[180] AND !F[179]) OR DI[26] OR DI[27])    ;
    :  DO[18181]=(OFF) ;
    :  F[329]=(OFF) ;
    :  F[298]=(F[180] OR F[179]) ;
    :  DO[1037]=(!DI[1037]) ;
    :  DO[18181]=(ON) ;
    :  WAIT ((DI[1037] AND !DI[1104]) OR (DI[1037] AND F[298]))    ;
    :  DO[18181]=(OFF) ;
    :  DO[1037]=(OFF) ;
    :  R[42]=33    ;
    :  !EZ3/SP3 wiederh. bei Messfehler ;
    :  IF (F[298]),JMP LBL[27] ;
    :  DO[1078]=(OFF) ;
    :  DO[1079]=(OFF) ;
    :  !KS nicht bei K-Verschleiss ;
    :  IF (DI[1097]),JMP LBL[35] ;
    :  !EZ3/SP3 2.Setzhub nach Fraesen ;
    :  IF (F[335] AND F[174]),JMP LBL[57] ;
    :  !EZ3/SP3 Kurzschluss schweissen ;
    :  IF (F[335] AND !F[174]),JMP LBL[34] ;
    :  !EZ3/SP3 Kurzschluss schweissen ;
    :  IF (!F[335]),JMP LBL[34] ;
    :   ;
    :  !************************** ;
    :  !*      Schritt 34        * ;
    :  !*     STAT EZ3/SP3       * ;
    :  !* Kurzschlussschweissung * ;
    :  !************************** ;
    :   ;
    :  LBL[34] ;
    :  R[41]=34    ;
    :  !RSK gestartet ;
    :  F[321]=(OFF) ;
    :  DO[209]=(ON) ;
    :  !EZ3/SP3/SK3 Prog. ;
    :  IF (F[174] AND !F[301]),GO[7]=(41) ;
    :  IF (F[174] AND !F[301]),GO[9]=(41) ;
    :  IF (F[175] OR F[301]),GO[7]=(51) ;
    :  IF (F[175] OR F[301]),GO[9]=(51) ;
    :  WAIT    .10(sec) ;
    :  DO[1037]=(OFF) ;
    :  DO[1038]=(OFF) ;
    :  DO[1105]=(OFF) ;
    :  DO[514]=(OFF) ;
    :  F[176]=(OFF) ;
    :  F[306]=(OFF) ;
    :  F[303]=(!DI[1089] AND DI[1104]) ;
    :  DO[18181]=(ON) ;
    :  WAIT (DI[1025] AND DI[1033] AND DI[1034] AND (!DI[1104] OR (DI[1089] AND DI[1104])))    ;
    :  DO[18181]=(OFF) ;
    :  F[303]=(OFF) ;
    :  DO[18181]=(ON) ;
    :  WAIT ((!DI[1105] AND DI[1112] AND DI[1122] AND !F[176]) OR (!DI[1112] AND DI[1122] AND DI[209]))    ;
    :  DO[18181]=(OFF) ;
    :  !EZ3/SP3 schliessen ;
    :  DO[1038]=(ON) ;
    :  TIMER[9]=((-4)) ;
    :  !EZ3/SP3 Kraft erreicht ;
    :  WAIT ((DI[1038] AND !DI[1092] AND !DI[1100]) OR DI[1094] OR DI[1095] OR (TIMER[9]>=0))    ;
    :  DO[1038]=(DI[1038] AND !DI[1094] AND !DI[1095]) ;
    :  DO[1037]=(!DO[1038]) ;
    :  !Schweissen START ;
    :  DO[1105]=(DI[1038] AND !DI[1094] AND !DI[1095]) ;
    :  !EZ3/SP3 Fehler Ausgleich ;
    :  F[302]=(DI[1038] AND DI[1039]) ;
    :  !EZ3/SP3 Fehler SZ ;
    :  F[300]=(DI[1094] OR DI[1095]) ;
    :  !SK3 FK ;
    :  TIMER[9]=((-10)) ;
    :  WAIT ((F[176] AND DO[1105]) OR ((DI[1124] OR DI[1125]) AND (DI[1105] AND DO[1105])) OR (DI[1091] AND DI[1104]) OR !DO[1105] OR (TIMER[9]>=0))    ;
    :  F[297]=(F[176] OR (DI[1124] AND !DI[1126] AND !DI[1095] AND DI[1105])) ;
    :  !SK3 Fehler ;
    :  F[301]=(!F[297] AND !F[298] AND DO[1105]) ;
    :  DO[1105]=(OFF) ;
    :  DO[1038]=(OFF) ;
    :  DO[18181]=(ON) ;
    :  F[749]=(!F[297] AND !F[748]) ;
    :  F[748]=(!F[297]) ;
    :  WAIT (F[297] OR DI[26] OR DI[27] OR (F[749] AND F[731]))    ;
    :  WAIT (!DI[26] AND !DI[27])    ;
    :  DO[18181]=(OFF) ;
    :  !EZ3/SP3 oeffnen ;
    :  DO[1037]=(!DI[1037]) ;
    :  DO[18181]=(ON) ;
    :  WAIT (DI[1037])    ;
    :  DO[18181]=(OFF) ;
    :  DO[1037]=(OFF) ;
    :  F[303]=(OFF) ;
    :  DO[209]=(OFF) ;
    :  R[42]=34    ;
    :  JMP LBL[35] ;
    :   ;
    :  !************************** ;
    :  !*       Schritt 35       * ;
    :  !*      STAT EZ3/SP3      * ;
    :  !************************** ;
    :   ;
    :  LBL[35] ;
    :  R[41]=35    ;
    :  !RSK gestartet ;
    :  F[321]=(OFF) ;
    :  !Sprung zurueck bei Fehler ;
    :  IF (!F[297] AND !DI[1097]),JMP LBL[27] ;
    :  !STAT EZ3/SP3 FK Fraesen ;
    :  F[185]=(!F[329]) ;
    :  DO[116]=(OFF) ;
    :  DO[194]=(OFF) ;
    :  R[42]=35    ;
    :  JMP LBL[1] ;
    :   ;
    :   ;
    :  !***************** ;
    :  !***************** ;
    :  !* MS1 Reinigung * ;
    :  !***************** ;
    :  !***************** ;
    :   ;
    :   ;
    :  !******************************* ;
    :  !*         Schritt 36          * ;
    :  !*       MS1 Reinigung         * ;
    :  !* KS3 in Arbeitsst. schwenken * ;
    :  !******************************* ;
    :   ;
    :  LBL[36] ;
    :  R[41]=36    ;
    :  !RSK gestartet ;
    :  F[321]=(OFF) ;
    :  !MS bei Reinigung ;
    :  DO[116]=(ON) ;
    :  !Reinigung MS1 gestartet ;
    :  F[604]=(ON) ;
    :  !Ueberwachungszeit KS3 ;
    :  TIMER[8]=((-4)) ;
    :  WAIT ((!DI[1164] AND DI[1162] AND DI[1165] AND !DI[1163]) OR (TIMER[8]>=0))    ;
    :  F[323]=((TIMER[8]>=0)) ;
    :  DO[18181]=((TIMER[8]>=0)) ;
    :  WAIT (!DI[1164] AND DI[1162] AND DI[1165] AND !DI[1163])    ;
    :  DO[18181]=(OFF) ;
    :  F[323]=(OFF) ;
    :  !KS3 in Arbeitsst. schwenken ;
    :  TIMER[8]=((-4)) ;
    :  DO[3974]=(ON) ;
    :  WAIT (DI[1161] OR (TIMER[8]>=0))    ;
    :  DO[18181]=((TIMER[8]>=0)) ;
    :  WAIT (DI[1161])    ;
    :  DO[18181]=(OFF) ;
    :  TIMER[8]=((-6)) ;
    :  WAIT ((DI[1164] AND !DI[1162] AND !DI[1165] AND DI[1163]) OR (TIMER[8]>=0))    ;
    :  F[324]=((TIMER[8]>=0)) ;
    :  DO[3974]=(OFF) ;
    :  DO[18181]=((TIMER[8]>=0)) ;
    :  WAIT ((DI[1164] AND !DI[1162] AND !DI[1165] AND DI[1163]) OR DI[26])    ;
    :  DO[18181]=(OFF) ;
    :  F[324]=(OFF) ;
    :  !Sprung bei Fehler KS3 schwenken ;
    :  IF (TIMER[8]>=0),JMP LBL[36] ;
    :  R[42]=36    ;
    :  JMP LBL[37] ;
    :   ;
    :  !*************************** ;
    :  !*      Schritt 37         * ;
    :  !* MS1 Reinigung starten   * ;
    :  !*************************** ;
    :   ;
    :  LBL[37] ;
    :  R[41]=37    ;
    :  TIMER[9]=((-2)) ;
    :  WAIT ((DI[10] AND DI[13] AND DI[23]) OR (TIMER[9]>=0))    ;
    :  F[329]=((TIMER[9]>=0)) ;
    :  DO[18181]=((TIMER[9]>=0)) ;
    :  WAIT (DI[10] AND DI[13] AND DI[23])    ;
    :  F[329]=(OFF) ;
    :  DO[18181]=(OFF) ;
    :  !MS1 Reinigung i.O. ;
    :  DO[18181]=(ON) ;
    :  WAIT (DI[1864])    ;
    :  DO[18181]=(OFF) ;
    :  !MS1 Ausblasen EIN ;
    :  DO[1870]=(ON) ;
    :  !MS1 Reinigung EIN ;
    :  TIMER[9]=((-1)) ;
    :  DO[1864]=(ON) ;
    :  !Einschaltdauer Reingung ;
    :  TIMER[7]=((R[26])) ;
    :  WAIT (!DI[1864] OR (TIMER[9]>=0))    ;
    :  F[329]=((TIMER[9]>=0)) ;
    :  DO[18181]=((TIMER[9]>=0)) ;
    :  WAIT (!DI[1864] OR DI[26])    ;
    :  WAIT ((TIMER[7]>=0))    ;
    :  F[329]=(OFF) ;
    :  DO[18181]=(OFF) ;
    :  !MS1 Reinigung AUS ;
    :  DO[1864]=(OFF) ;
    :  TIMER[9]=((-6)) ;
    :  WAIT (DI[1864] OR (TIMER[9]>=0))    ;
    :  F[329]=((TIMER[9]>=0)) ;
    :  DO[18181]=((TIMER[9]>=0)) ;
    :  WAIT (DI[1864] OR DI[26] OR !DI[13] OR !DI[23])    ;
    :  IF (DI[26] OR !DI[13] OR !DI[23]),JMP LBL[37] ;
    :  F[329]=(OFF) ;
    :  DO[18181]=(OFF) ;
    :  !MS1 Ausblasen AUS ;
    :  DO[1870]=(OFF) ;
    :  !MS1 Einspruehen ;
    :  TIMER[9]=((R[23])) ;
    :  DO[520]=(!F[574] AND F[575]) ;
    :  DO[1871]=(F[574] AND F[575]) ;
    :  WAIT (!F[575] OR (TIMER[9]>=0))    ;
    :  DO[520]=(OFF) ;
    :  DO[1871]=(OFF) ;
    :  R[42]=37    ;
    :  JMP LBL[38] ;
    :   ;
    :  !**************************** ;
    :  !*          Schritt 38      * ;
    :  !*       MS1 Reinigung      * ;
    :  !* KS3 in Ruhest. schwenken * ;
    :  !**************************** ;
    :   ;
    :  LBL[38] ;
    :  R[41]=38    ;
    :  !Ueberwachungszeit KS3 ;
    :  TIMER[8]=((-4)) ;
    :  WAIT ((DI[1164] AND !DI[1162] AND !DI[1165] AND DI[1163]) OR (TIMER[8]>=0))    ;
    :  F[324]=((TIMER[8]>=0)) ;
    :  DO[18181]=((TIMER[8]>=0)) ;
    :  WAIT (DI[1164] AND !DI[1162] AND !DI[1165] AND DI[1163])    ;
    :  DO[18181]=(OFF) ;
    :  F[324]=(OFF) ;
    :  !KS3 in Ruhestest. schwenken ;
    :  TIMER[8]=((-4)) ;
    :  DO[3971]=(ON) ;
    :  WAIT (DI[1161] OR (TIMER[8]>=0))    ;
    :  DO[18181]=((TIMER[8]>=0)) ;
    :  WAIT (DI[1161])    ;
    :  DO[18181]=(OFF) ;
    :  TIMER[8]=((-6)) ;
    :  WAIT ((!DI[1164] AND DI[1162] AND DI[1165] AND !DI[1163]) OR (TIMER[8]>=0))    ;
    :  F[323]=((TIMER[8]>=0)) ;
    :  DO[3971]=(OFF) ;
    :  DO[18181]=((TIMER[8]>=0)) ;
    :  WAIT ((!DI[1164] AND DI[1162] AND DI[1165] AND !DI[1163]) OR DI[26])    ;
    :  DO[18181]=(OFF) ;
    :  F[323]=(OFF) ;
    :  !Sprung bei Fehler KS3 schwenken ;
    :  IF (TIMER[8]>=0),JMP LBL[38] ;
    :  R[42]=38    ;
    :  JMP LBL[39] ;
    :   ;
    :  !***************************** ;
    :  !*         Schritt 39        * ;
    :  !* MS1 Reinigung ruecksetzen * ;
    :  !***************************** ;
    :   ;
    :  LBL[39] ;
    :  R[41]=39    ;
    :  !MS1 Zaehler ruecksetzen ;
    :  R[21]=0    ;
    :  !MS FRG Reinigung ;
    :  F[603]=(OFF) ;
    :  !MS1 Reinigung FK ;
    :  F[605]=(ON) ;
    :  R[42]=39    ;
    :  JMP LBL[1] ;
    :   ;
    :   ;
    :  !***************** ;
    :  !***************** ;
    :  !* MS2 Reinigung * ;
    :  !***************** ;
    :  !***************** ;
    :   ;
    :   ;
    :  !******************************* ;
    :  !*         Schritt 40          * ;
    :  !*       MS2 Reinigung         * ;
    :  !* KS2 in Arbeitsst. schwenken * ;
    :  !******************************* ;
    :   ;
    :  LBL[40] ;
    :  R[41]=40    ;
    :  !RSK gestartet ;
    :  F[321]=(OFF) ;
    :  !Reinigung MS2 gestartet ;
    :  F[608]=(ON) ;
    :  !MS bei Reinigung ;
    :  DO[116]=(ON) ;
    :  !Ueberwachungszeit KS2 ;
    :  TIMER[8]=((-4)) ;
    :  WAIT ((!DI[1004] AND DI[1002] AND DI[1005] AND !DI[1003]) OR (TIMER[8]>=0))    ;
    :  F[323]=((TIMER[8]>=0)) ;
    :  DO[18181]=((TIMER[8]>=0)) ;
    :  WAIT (!DI[1004] AND DI[1002] AND DI[1005] AND !DI[1003])    ;
    :  DO[18181]=(OFF) ;
    :  F[323]=(OFF) ;
    :  !KS2 in Arbeitsst. schwenken ;
    :  TIMER[8]=((-4)) ;
    :  DO[3973]=(ON) ;
    :  WAIT (DI[1001] OR (TIMER[8]>=0))    ;
    :  DO[18181]=((TIMER[8]>=0)) ;
    :  WAIT (DI[1001])    ;
    :  DO[18181]=(OFF) ;
    :  TIMER[8]=((-4)) ;
    :  WAIT ((DI[1004] AND !DI[1002] AND !DI[1005] AND DI[1003]) OR (TIMER[8]>=0))    ;
    :  F[324]=((TIMER[8]>=0)) ;
    :  DO[3973]=(OFF) ;
    :  DO[18181]=((TIMER[8]>=0)) ;
    :  WAIT ((DI[1004] AND !DI[1002] AND !DI[1005] AND DI[1003]) OR DI[26])    ;
    :  DO[18181]=(OFF) ;
    :  F[324]=(OFF) ;
    :  !Sprung bei Fehler KS2 schwenken ;
    :  IF (TIMER[8]>=0),JMP LBL[40] ;
    :  R[42]=40    ;
    :  JMP LBL[41] ;
    :   ;
    :  !*************************** ;
    :  !*      Schritt 41         * ;
    :  !* MS2 Reinigung starten   * ;
    :  !*************************** ;
    :   ;
    :  LBL[41] ;
    :  R[41]=41    ;
    :  TIMER[9]=((-2)) ;
    :  WAIT ((DI[10] AND DI[13] AND DI[23]) OR (TIMER[9]>=0))    ;
    :  F[329]=((TIMER[9]>=0)) ;
    :  DO[18181]=((TIMER[9]>=0)) ;
    :  WAIT (DI[10] AND DI[13] AND DI[23])    ;
    :  F[329]=(OFF) ;
    :  DO[18181]=(OFF) ;
    :  !MS2 Ausblasen EIN ;
    :  DO[1902]=(ON) ;
    :  !MS2 Reinigung EIN ;
    :  TIMER[9]=((-1)) ;
    :  DO[1896]=(ON) ;
    :  WAIT (!DI[1896] OR (TIMER[9]>=0))    ;
    :  F[329]=((TIMER[9]>=0)) ;
    :  DO[18181]=((TIMER[9]>=0)) ;
    :  WAIT (!DI[1896] OR DI[26])    ;
    :  F[329]=(OFF) ;
    :  DO[18181]=(OFF) ;
    :  !MS2 Reinigung AUS ;
    :  DO[1896]=(OFF) ;
    :  TIMER[9]=((-6)) ;
    :  WAIT (DI[1896] OR (TIMER[9]>=0))    ;
    :  F[329]=((TIMER[9]>=0)) ;
    :  DO[18181]=((TIMER[9]>=0)) ;
    :  WAIT (DI[1896] OR DI[26] OR !DI[13] OR !DI[23])    ;
    :  IF (DI[26] OR !DI[13] OR !DI[23]),JMP LBL[41] ;
    :  F[329]=(OFF) ;
    :  DO[18181]=(OFF) ;
    :  !MS2 Ausblasen AUS ;
    :  DO[1902]=(OFF) ;
    :  !MS2 Einspruehen ;
    :  TIMER[9]=((R[23])) ;
    :  DO[528]=(!F[583] AND F[584]) ;
    :  DO[1903]=(F[583] AND F[585]) ;
    :  WAIT (!F[584] OR (TIMER[9]>=0))    ;
    :  DO[528]=(OFF) ;
    :  DO[1903]=(OFF) ;
    :  R[42]=41    ;
    :  JMP LBL[42] ;
    :   ;
    :  !**************************** ;
    :  !*          Schritt 42      * ;
    :  !*       MS2 Reinigung      * ;
    :  !* KS2 in Ruhest. schwenken * ;
    :  !**************************** ;
    :   ;
    :  LBL[42] ;
    :  R[41]=42    ;
    :  !Ueberwachungszeit KS2 ;
    :  TIMER[8]=((-4)) ;
    :  WAIT ((DI[1004] AND !DI[1002] AND !DI[1005] AND DI[1003]) OR (TIMER[8]>=0))    ;
    :  F[324]=((TIMER[8]>=0)) ;
    :  DO[18181]=((TIMER[8]>=0)) ;
    :  WAIT (DI[1004] AND !DI[1002] AND !DI[1005] AND DI[1003])    ;
    :  DO[18181]=(OFF) ;
    :  F[324]=(OFF) ;
    :  !KS2 in Ruhestest. schwenken ;
    :  TIMER[8]=((-4)) ;
    :  DO[3970]=(ON) ;
    :  WAIT (DI[1001] OR (TIMER[8]>=0))    ;
    :  DO[18181]=((TIMER[8]>=0)) ;
    :  WAIT (DI[1001])    ;
    :  DO[18181]=(OFF) ;
    :  TIMER[8]=((-6)) ;
    :  WAIT ((!DI[1004] AND DI[1002] AND DI[1005] AND !DI[1003]) OR (TIMER[8]>=0))    ;
    :  F[323]=((TIMER[8]>=0)) ;
    :  DO[3970]=(OFF) ;
    :  DO[18181]=((TIMER[8]>=0)) ;
    :  WAIT ((!DI[1004] AND DI[1002] AND DI[1005] AND !DI[1003]) OR DI[26])    ;
    :  DO[18181]=(OFF) ;
    :  F[323]=(OFF) ;
    :  !Sprung bei Fehler KS2 schwenken ;
    :  IF (TIMER[8]>=0),JMP LBL[42] ;
    :  R[42]=42    ;
    :  JMP LBL[43] ;
    :   ;
    :  !***************************** ;
    :  !*         Schritt 43        * ;
    :  !* MS2 Reinigung ruecksetzen * ;
    :  !***************************** ;
    :   ;
    :  LBL[43] ;
    :  R[41]=43    ;
    :  !MS2 Zaehler ruecksetzen ;
    :  R[22]=0    ;
    :  !MS2 FRG Reinigung ;
    :  F[607]=(OFF) ;
    :  !MS2 Reinigung FK ;
    :  F[609]=(ON) ;
    :  R[42]=43    ;
    :  JMP LBL[1] ;
    :   ;
    :  !******************************** ;
    :  !*            Schritt 44 ;
    :  !*          KL1 Spueleimer ;
    :  !*  (an Pneum. Schwenkeinheit KL1 ;
    :  !*     KL1 in Arbeitsst. schwenke ;
    :  !******************************** ;
    :   ;
    :  LBL[44] ;
    :  R[41]=44    ;
    :  !RSK gestartet ;
    :  F[321]=(OFF) ;
    :  DO[161]=(ON) ;
    :  !Steuerluft EIN ;
    :  DO[2113]=(ON) ;
    :  TIMER[9]=((-2)) ;
    :  !Warte auf Vorwahl Ventilinsel ;
    :  WAIT ((F[523] AND !F[524]) OR (!F[523] AND F[524]) OR (TIMER[9]>=0))    ;
    :  DO[120]=(TIMER[9]>=0) ;
    :  DO[18181]=((TIMER[9]>=0)) ;
    :  WAIT ((F[523] AND !F[524]) OR (!F[523] AND F[524]))    ;
    :  DO[120]=(OFF) ;
    :  DO[18181]=(OFF) ;
    :  !WAIT Steuerluft EIN ;
    :  WAIT ((F[523] AND !F[524] AND DI[2113]) OR (!F[523] AND F[524] AND !DI[2114]) OR (TIMER[9]>=0))    ;
    :  DO[120]=(TIMER[9]>=0) ;
    :  DO[18181]=((TIMER[9]>=0)) ;
    :  WAIT ((F[523] AND !F[524] AND DI[2113]) OR (!F[523] AND F[524] AND !DI[2114]))    ;
    :  DO[120]=(OFF) ;
    :  DO[18181]=(OFF) ;
    :  !In Arbeitsstellung schwenken ;
    :  DO[2115]=(OFF) ;
    :  DO[2116]=(ON) ;
    :  !Freigabe Bewegung (ON) ;
    :  DO[2117]=(OFF) ;
    :  DO[2118]=(ON) ;
    :  TIMER[9]=((-10)) ;
    :  !Warte bis Spueleimer in Position ;
    :  WAIT ((!DI[2115] AND DI[2116]) OR (TIMER[9]>=0))    ;
    :  DO[120]=(TIMER[9]>=0) ;
    :  DO[18181]=((TIMER[9]>=0)) ;
    :  WAIT (!DI[2115] AND DI[2116])    ;
    :  DO[120]=(OFF) ;
    :  DO[18181]=(OFF) ;
    :  F[355]=((!DI[2115] AND DI[2116]) OR (F[837])) ;
    :  WAIT    .30(sec) ;
    :  !In Ruhestellung schwenken AUS ;
    :  DO[2115]=(OFF) ;
    :  !In Arbeitsstellung schw. AUS ;
    :  DO[2116]=(OFF) ;
    :  !Freigabe Bewegung AUS ;
    :  DO[2118]=(OFF) ;
    :  TIMER[9]=((-5)) ;
    :  WAIT ((DI[2118]) OR (DI[2117] AND F[837]) OR (TIMER[9]>=0))    ;
    :  DO[120]=(TIMER[9]>=0) ;
    :  DO[18181]=((TIMER[9]>=0)) ;
    :  WAIT ((DI[2118]) OR (DI[2117] AND F[837]))    ;
    :  DO[120]=(OFF) ;
    :  DO[18181]=(OFF) ;
    :  !Freigabe  in  Endlage  halten ;
    :  DO[2117]=(!F[837]) ;
    :  IF (F[837]),DO[2118]=PULSE,0.5sec ;
    :  TIMER[9]=((-10)) ;
    :  WAIT ((DI[2117]) OR (DI[2118] AND F[837]) OR (TIMER[9]>=0))    ;
    :  DO[120]=(TIMER[9]>=0) ;
    :  DO[18181]=((TIMER[9]>=0)) ;
    :  WAIT ((DI[2117]) OR (DI[2118] AND F[837]))    ;
    :  DO[120]=(OFF) ;
    :  DO[18181]=(OFF) ;
    :  DO[161]=(OFF) ;
    :  R[42]=44    ;
    :  JMP LBL[1] ;
    :   ;
    :  !******************************** ;
    :  !*           Schritt 45 ;
    :  !*         KL1 Spueleimer ;
    :  !* (an Pneum. Schwenkeinheit KL1) ;
    :  !*    KL1 in Ruhest. schwenken ;
    :  !******************************** ;
    :   ;
    :  LBL[45] ;
    :  R[41]=45    ;
    :  !RSK gestartet ;
    :  F[321]=(OFF) ;
    :  DO[161]=(ON) ;
    :  !Steuerluft EIN ;
    :  DO[2113]=(ON) ;
    :  TIMER[9]=((-2)) ;
    :  !Warte auf Vorwahl Ventilinsel ;
    :  WAIT ((F[523] AND !F[524]) OR (!F[523] AND F[524]) OR (TIMER[9]>=0))    ;
    :  DO[120]=(TIMER[9]>=0) ;
    :  DO[18181]=((TIMER[9]>=0)) ;
    :  WAIT ((F[523] AND !F[524]) OR (!F[523] AND F[524]))    ;
    :  DO[120]=(OFF) ;
    :  DO[18181]=(OFF) ;
    :  !Warte bis Steuerluft EIN ;
    :  WAIT ((F[523] AND !F[524] AND DI[2113]) OR (!F[523] AND F[524] AND !DI[2114]) OR (TIMER[9]>=0))    ;
    :  DO[120]=(TIMER[9]>=0) ;
    :  DO[18181]=((TIMER[9]>=0)) ;
    :  WAIT ((F[523] AND !F[524] AND DI[2113]) OR (!F[523] AND F[524] AND !DI[2114]))    ;
    :  DO[120]=(OFF) ;
    :  DO[18181]=(OFF) ;
    :  !In Ruhestellung schwenken EIN ;
    :  DO[2115]=(ON) ;
    :  DO[2116]=(OFF) ;
    :  !Freigabe Bewegung EIN ;
    :  DO[2117]=(OFF) ;
    :  DO[2118]=(ON) ;
    :  TIMER[9]=((-10)) ;
    :  !Warte bis Spueleimer in Position ;
    :  WAIT ((DI[2115] AND !DI[2116]) OR (TIMER[9]>=0))    ;
    :  DO[120]=(TIMER[9]>=0) ;
    :  DO[18181]=((TIMER[9]>=0)) ;
    :  WAIT (DI[2115] AND !DI[2116])    ;
    :  DO[120]=(OFF) ;
    :  DO[18181]=(OFF) ;
    :  F[355]=((DI[2115] AND !DI[2116]) OR (F[837])) ;
    :  WAIT    .30(sec) ;
    :  !In Ruhestellung schwenken AUS ;
    :  DO[2115]=(OFF) ;
    :  !In Arbeitsstellung schw. AUS ;
    :  DO[2116]=(OFF) ;
    :  !Freigabe Bewegung AUS ;
    :  DO[2118]=(OFF) ;
    :  TIMER[9]=((-5)) ;
    :  WAIT ((DI[2118]) OR (DI[2117] AND F[837]) OR (TIMER[9]>=0))    ;
    :  DO[120]=(TIMER[9]>=0) ;
    :  DO[18181]=((TIMER[9]>=0)) ;
    :  WAIT ((DI[2118]) OR (DI[2117] AND F[837]))    ;
    :  DO[120]=(OFF) ;
    :  DO[18181]=(OFF) ;
    :  !Freigabe  in  Endlage  halten ;
    :  DO[2117]=(!F[837]) ;
    :  IF (F[837]),DO[2118]=PULSE,0.5sec ;
    :  TIMER[9]=((-10)) ;
    :  WAIT ((DI[2117]) OR (DI[2118] AND F[837]) OR (TIMER[9]>=0))    ;
    :  DO[120]=(TIMER[9]>=0) ;
    :  DO[18181]=((TIMER[9]>=0)) ;
    :  WAIT ((DI[2117]) OR (DI[2118] AND F[837]))    ;
    :  DO[120]=(OFF) ;
    :  DO[18181]=(OFF) ;
    :  DO[161]=(OFF) ;
    :  R[42]=45    ;
    :  JMP LBL[1] ;
    :   ;
    :  !******************************** ;
    :  !*            Schritt 46 ;
    :  !*          KL2 Spueleimer ;
    :  !*  (an Pneum. Schwenkeinheit KL2 ;
    :  !*     KL2 in Arbeitsst. schwenke ;
    :  !******************************** ;
    :   ;
    :  LBL[46] ;
    :  R[41]=46    ;
    :  !RSK gestartet ;
    :  F[321]=(OFF) ;
    :  DO[177]=(ON) ;
    :  !Steuerluft EIN ;
    :  DO[2121]=(ON) ;
    :  TIMER[9]=((-2)) ;
    :  !Warte auf Vorwahl Ventilinsel ;
    :  WAIT ((F[523] AND !F[524]) OR (!F[523] AND F[524]) OR (TIMER[9]>=0))    ;
    :  DO[120]=(TIMER[9]>=0) ;
    :  DO[18181]=((TIMER[9]>=0)) ;
    :  WAIT ((F[523] AND !F[524]) OR (!F[523] AND F[524]))    ;
    :  DO[120]=(OFF) ;
    :  DO[18181]=(OFF) ;
    :  !Warte Steuerluft EIN ;
    :  WAIT ((F[523] AND !F[524] AND DI[2121]) OR (!F[523] AND F[524] AND !DI[2122]) OR (TIMER[9]>=0))    ;
    :  DO[120]=(TIMER[9]>=0) ;
    :  DO[18181]=((TIMER[9]>=0)) ;
    :  WAIT ((F[523] AND !F[524] AND DI[2121]) OR (!F[523] AND F[524] AND !DI[2122]))    ;
    :  DO[120]=(OFF) ;
    :  DO[18181]=(OFF) ;
    :  !In Arbeitsstellung schwenken EI ;
    :  DO[2123]=(OFF) ;
    :  DO[2124]=(ON) ;
    :  !Freigabe Bewegung EIN ;
    :  DO[2125]=(OFF) ;
    :  DO[2126]=(ON) ;
    :  TIMER[9]=((-10)) ;
    :  !Warte bis Spueleimer in Position ;
    :  WAIT ((!DI[2123] AND DI[2124]) OR (TIMER[9]>=0))    ;
    :  DO[120]=(TIMER[9]>=0) ;
    :  DO[18181]=((TIMER[9]>=0)) ;
    :  WAIT (!DI[2123] AND DI[2124])    ;
    :  DO[120]=(OFF) ;
    :  DO[18181]=(OFF) ;
    :  F[376]=(!DI[2123] AND DI[2124]) ;
    :  WAIT    .30(sec) ;
    :  !In Ruhestellung schwenken AUS ;
    :  DO[2123]=(OFF) ;
    :  !In Arbeitsstellung schwenken AU ;
    :  DO[2124]=(OFF) ;
    :  !Freigabe Bewegung AUS ;
    :  DO[2126]=(OFF) ;
    :  TIMER[9]=((-5)) ;
    :  WAIT (DI[2126] OR (TIMER[9]>=0))    ;
    :  DO[120]=(TIMER[9]>=0) ;
    :  DO[18181]=((TIMER[9]>=0)) ;
    :  WAIT (DI[2126])    ;
    :  DO[120]=(OFF) ;
    :  DO[18181]=(OFF) ;
    :  !Freigabe  in  Endlage  halten ;
    :  DO[2125]=(ON) ;
    :  TIMER[9]=((-10)) ;
    :  WAIT (DI[2125] OR (TIMER[9]>=0))    ;
    :  DO[120]=(TIMER[9]>=0) ;
    :  DO[18181]=((TIMER[9]>=0)) ;
    :  WAIT (DI[2125])    ;
    :  DO[120]=(OFF) ;
    :  DO[18181]=(OFF) ;
    :  DO[177]=(OFF) ;
    :  R[42]=46    ;
    :  JMP LBL[1] ;
    :   ;
    :  !******************************** ;
    :  !*           Schritt 47 ;
    :  !*         KL2 Spueleimer ;
    :  !* (an Pneum. Schwenkeinheit KL2) ;
    :  !*    KL2 in Ruhest. schwenken ;
    :  !******************************** ;
    :   ;
    :  LBL[47] ;
    :  R[41]=47    ;
    :  !RSK gestartet ;
    :  F[321]=(OFF) ;
    :  DO[177]=(ON) ;
    :  !Steuerluft EIN ;
    :  DO[2121]=(ON) ;
    :  TIMER[9]=((-2)) ;
    :  !Warte auf Vorwahl Ventilinsel ;
    :  WAIT ((F[523] AND !F[524]) OR (!F[523] AND F[524]) OR (TIMER[9]>=0))    ;
    :  DO[120]=(TIMER[9]>=0) ;
    :  DO[18181]=((TIMER[9]>=0)) ;
    :  WAIT ((F[523] AND !F[524]) OR (!F[523] AND F[524]))    ;
    :  DO[120]=(OFF) ;
    :  DO[18181]=(OFF) ;
    :  !Warte Steuerluft EIN ;
    :  WAIT ((F[523] AND !F[524] AND DI[2121]) OR (!F[523] AND F[524] AND !DI[2122]) OR (TIMER[9]>=0))    ;
    :  DO[120]=(TIMER[9]>=0) ;
    :  DO[18181]=((TIMER[9]>=0)) ;
    :  WAIT ((F[523] AND !F[524] AND DI[2121]) OR (!F[523] AND F[524] AND !DI[2122]))    ;
    :  DO[120]=(OFF) ;
    :  DO[18181]=(OFF) ;
    :  !In Ruhestellung schwenken EIN ;
    :  DO[2123]=(ON) ;
    :  DO[2124]=(OFF) ;
    :  !Freigabe Bewegung EIN ;
    :  DO[2125]=(OFF) ;
    :  DO[2126]=(ON) ;
    :  TIMER[9]=((-10)) ;
    :  !Warte bis Spueleimer in Position ;
    :  WAIT ((DI[2123] AND !DI[2124]) OR (TIMER[9]>=0))    ;
    :  DO[120]=(TIMER[9]>=0) ;
    :  DO[18181]=((TIMER[9]>=0)) ;
    :  WAIT (DI[2123] AND !DI[2124])    ;
    :  DO[120]=(OFF) ;
    :  DO[18181]=(OFF) ;
    :  F[376]=(DI[2123] AND !DI[2124]) ;
    :  WAIT    .30(sec) ;
    :  !In Ruhestellung schwenken AUS ;
    :  DO[2123]=(OFF) ;
    :  !In Arbeitsstellung schwenken AU ;
    :  DO[2124]=(OFF) ;
    :  !Freigabe Bewegung AUS ;
    :  DO[2126]=(OFF) ;
    :  TIMER[9]=((-5)) ;
    :  WAIT (DI[2126] OR (TIMER[9]>=0))    ;
    :  DO[120]=(TIMER[9]>=0) ;
    :  DO[18181]=((TIMER[9]>=0)) ;
    :  WAIT (DI[2126])    ;
    :  DO[120]=(OFF) ;
    :  DO[18181]=(OFF) ;
    :  !Freigabe  in  Endlage  halten ;
    :  DO[2125]=(ON) ;
    :  TIMER[9]=((-10)) ;
    :  WAIT (DI[2125] OR (TIMER[9]>=0))    ;
    :  DO[120]=(TIMER[9]>=0) ;
    :  DO[18181]=((TIMER[9]>=0)) ;
    :  WAIT (DI[2125])    ;
    :  DO[120]=(OFF) ;
    :  DO[18181]=(OFF) ;
    :  DO[177]=(OFF) ;
    :  R[42]=47    ;
    :  JMP LBL[1] ;
    :   ;
    :  !******************************** ;
    :  !*            Schritt 48 ;
    :  !*          KL3 Spueleimer ;
    :  !*  (an Pneum. Schwenkeinheit KL3 ;
    :  !*     KL3 in Arbeitsst. schwenke ;
    :  !******************************** ;
    :   ;
    :  LBL[48] ;
    :  R[41]=48    ;
    :  !RSK gestartet ;
    :  F[321]=(OFF) ;
    :  DO[193]=(ON) ;
    :  !Steuerluft EIN ;
    :  DO[2129]=(ON) ;
    :  TIMER[9]=((-2)) ;
    :  !Warte auf Vorwahl Ventilinsel ;
    :  WAIT ((F[523] AND !F[524]) OR (!F[523] AND F[524]) OR (TIMER[9]>=0))    ;
    :  DO[120]=(TIMER[9]>=0) ;
    :  DO[18181]=((TIMER[9]>=0)) ;
    :  WAIT ((F[523] AND !F[524]) OR (!F[523] AND F[524]))    ;
    :  DO[120]=(OFF) ;
    :  DO[18181]=(OFF) ;
    :  !Warte bis Steuerluft EIN ;
    :  WAIT ((F[523] AND !F[524] AND DI[2129]) OR (!F[523] AND F[524] AND !DI[2130]) OR (TIMER[9]>=0))    ;
    :  DO[120]=(TIMER[9]>=0) ;
    :  DO[18181]=((TIMER[9]>=0)) ;
    :  WAIT ((F[523] AND !F[524] AND DI[2129]) OR (!F[523] AND F[524] AND !DI[2130]))    ;
    :  DO[120]=(OFF) ;
    :  DO[18181]=(OFF) ;
    :  !In Arbeitsstellung schwenken EI ;
    :  DO[2131]=(OFF) ;
    :  DO[2132]=(ON) ;
    :  !Freigabe Bewegung EIN ;
    :  DO[2133]=(OFF) ;
    :  DO[2134]=(ON) ;
    :  TIMER[9]=((-10)) ;
    :  !Warte bis Spueleimer in Position ;
    :  WAIT ((!DI[2131] AND DI[2132]) OR (TIMER[9]>=0))    ;
    :  DO[120]=(TIMER[9]>=0) ;
    :  DO[18181]=((TIMER[9]>=0)) ;
    :  WAIT (!DI[2131] AND DI[2132])    ;
    :  DO[120]=(OFF) ;
    :  DO[18181]=(OFF) ;
    :  F[397]=(!DI[2131] AND DI[2132]) ;
    :  WAIT    .30(sec) ;
    :  !In Ruhestellung schwenken AUS ;
    :  DO[2131]=(OFF) ;
    :  ! In Arbeitsstellung schwenken A ;
    :  DO[2132]=(OFF) ;
    :  !Freigabe Bewegung AUS ;
    :  DO[2134]=(OFF) ;
    :  TIMER[9]=((-5)) ;
    :  WAIT (DI[2134] OR (TIMER[9]>=0))    ;
    :  DO[120]=(TIMER[9]>=0) ;
    :  DO[18181]=((TIMER[9]>=0)) ;
    :  WAIT (DI[2134])    ;
    :  DO[120]=(OFF) ;
    :  DO[18181]=(OFF) ;
    :  !Freigabe  in  Endlage  halten ;
    :  DO[2133]=(ON) ;
    :  TIMER[9]=((-10)) ;
    :  WAIT (DI[2133] OR (TIMER[9]>=0))    ;
    :  DO[120]=(TIMER[9]>=0) ;
    :  DO[18181]=((TIMER[9]>=0)) ;
    :  WAIT (DI[2133])    ;
    :  DO[120]=(OFF) ;
    :  DO[18181]=(OFF) ;
    :  DO[193]=(OFF) ;
    :  R[42]=48    ;
    :  JMP LBL[1] ;
    :   ;
    :  !******************************** ;
    :  !*           Schritt 49 ;
    :  !*         KL3 Spueleimer ;
    :  !* (an Pneum. Schwenkeinheit KL3) ;
    :  !*    KL3 in Ruhest. schwenken ;
    :  !******************************** ;
    :   ;
    :  LBL[49] ;
    :  R[41]=49    ;
    :  !RSK gestartet ;
    :  F[321]=(OFF) ;
    :  DO[193]=(ON) ;
    :  !Steuerluft EIN ;
    :  DO[2129]=(ON) ;
    :  TIMER[9]=((-2)) ;
    :  !Warte auf Vorwahl Ventilinsel ;
    :  WAIT ((F[523] AND !F[524]) OR (!F[523] AND F[524]) OR (TIMER[9]>=0))    ;
    :  DO[120]=(TIMER[9]>=0) ;
    :  DO[18181]=((TIMER[9]>=0)) ;
    :  WAIT ((F[523] AND !F[524]) OR (!F[523] AND F[524]))    ;
    :  DO[120]=(OFF) ;
    :  DO[18181]=(OFF) ;
    :  !Warte bis Steuerluft EIN ;
    :  WAIT ((F[523] AND !F[524] AND DI[2129]) OR (!F[523] AND F[524] AND !DI[2130]) OR (TIMER[9]>=0))    ;
    :  DO[120]=(TIMER[9]>=0) ;
    :  DO[18181]=((TIMER[9]>=0)) ;
    :  WAIT ((F[523] AND !F[524] AND DI[2129]) OR (!F[523] AND F[524] AND !DI[2130]))    ;
    :  DO[120]=(OFF) ;
    :  DO[18181]=(OFF) ;
    :  !In Ruhestellung schwenken EI ;
    :  DO[2131]=(ON) ;
    :  DO[2132]=(OFF) ;
    :  !Freigabe Bewegung EIN ;
    :  DO[2133]=(OFF) ;
    :  DO[2134]=(ON) ;
    :  TIMER[9]=((-10)) ;
    :  !Warte bis Spueleimer in Position ;
    :  WAIT ((DI[2131] AND !DI[2132]) OR (TIMER[9]>=0))    ;
    :  DO[120]=(TIMER[9]>=0) ;
    :  DO[18181]=((TIMER[9]>=0)) ;
    :  WAIT (DI[2131] AND DI[2132])    ;
    :  DO[120]=(OFF) ;
    :  DO[18181]=(OFF) ;
    :  F[397]=(DI[2131] AND !DI[2132]) ;
    :  WAIT    .30(sec) ;
    :  !In Ruhestellung schwenken AUS ;
    :  DO[2131]=(OFF) ;
    :  !In Arbeitsstellung schwenken A ;
    :  DO[2132]=(OFF) ;
    :  !Freigabe Bewegung AUS ;
    :  DO[2134]=(OFF) ;
    :  TIMER[9]=((-5)) ;
    :  WAIT (DI[2134] OR (TIMER[9]>=0))    ;
    :  DO[120]=(TIMER[9]>=0) ;
    :  DO[18181]=((TIMER[9]>=0)) ;
    :  WAIT (DI[2134])    ;
    :  DO[120]=(OFF) ;
    :  DO[18181]=(OFF) ;
    :  !Freigabe  in  Endlage  halten ;
    :  DO[2133]=(ON) ;
    :  TIMER[9]=((-10)) ;
    :  WAIT (DI[2133] OR (TIMER[9]>=0))    ;
    :  DO[120]=(TIMER[9]>=0) ;
    :  DO[18181]=((TIMER[9]>=0)) ;
    :  WAIT (DI[2133])    ;
    :  DO[120]=(OFF) ;
    :  DO[18181]=(OFF) ;
    :  DO[193]=(OFF) ;
    :  R[42]=49    ;
    :  JMP LBL[1] ;
    :   ;
    :   ;
    :  !********************** ;
    :  !*    MS1 Reinigung   * ;
    :  !*     (an Pneum. )   * ;
    :  !* Schwenkeinheit MS1 * ;
    :  !********************** ;
    :   ;
    :   ;
    :  !******************************* ;
    :  !*         Schritt 50          * ;
    :  !*       MS1 Reinigung         * ;
    :  !* MS1 in Arbeitsst. schwenken * ;
    :  !******************************* ;
    :   ;
    :  LBL[50] ;
    :  R[41]=50    ;
    :  !RSK gestartet ;
    :  F[321]=(OFF) ;
    :  F[323]=(OFF) ;
    :  F[324]=(OFF) ;
    :  F[329]=(OFF) ;
    :  !Reinigung MS1 gestartet ;
    :  !MS bei Reinigung ;
    :  DO[116]=(ON) ;
    :  !Reinigung MS1 gestartet ;
    :  F[604]=(ON) ;
    :  !Steuerluft EIN ;
    :  DO[2161]=(ON) ;
    :  DO[2163]=(OFF) ;
    :  DO[2164]=(OFF) ;
    :  DO[2165]=(OFF) ;
    :  DO[2166]=(OFF) ;
    :  DO[2167]=(OFF) ;
    :  DO[2168]=(OFF) ;
    :  !Ueberwachungszeit Schwenkeinheit ;
    :  TIMER[8]=((-5)) ;
    :  !RSK Fehlerausgabe Schwenkeinheit ;
    :  F[323]=(!DI[2163]) ;
    :  !RSK Sammelstoerung ;
    :  F[329]=(F[323]) ;
    :  !Sprung bei Fehler MS1 schwenken ;
    :  IF ((DI[26] OR DI[27]) AND F[323]),JMP LBL[50] ;
    :  WAIT ((!F[323] OR (TIMER[8]>=0)) AND ((F[523] AND !F[524] AND DI[2161]) OR (!F[523] AND F[524] AND !DI[2162])))    ;
    :  !Schwenkeinheit 1 in Arbeitsstell ;
    :  DO[2163]=(OFF) ;
    :  DO[2164]=(!DO[2164]) ;
    :  !FRG Bewegung EIN ;
    :  DO[2165]=(OFF) ;
    :  DO[2166]=(!DI[2164]) ;
    :  DO[18181]=(ON) ;
    :  WAIT ((DI[2164] AND !DI[2163]) OR (TIMER[8]>=0))    ;
    :  DO[18181]=(OFF) ;
    :  !RSK Fehlerausgabe Schwenkeinheit ;
    :  F[324]=((!DI[2164] AND (TIMER[8]>=0)) OR F[324]) ;
    :  !RSK Sammelstoerung ;
    :  F[329]=(F[324]) ;
    :  !In Ruhestellung schwenken AUS ;
    :  DO[2163]=(OFF) ;
    :  !In Arbeitsstellung schwenken AUS ;
    :  DO[2164]=(OFF) ;
    :  !FRG Bewegung AUS ;
    :  DO[2166]=(OFF) ;
    :  IF ((DI[26] OR DI[27]) AND F[324]),JMP LBL[50] ;
    :  IF (!F[324] AND DI[2166]),JMP LBL[51] ;
    :   ;
    :  !*************************** ;
    :  !*      Schritt 51         * ;
    :  !*  MS1 Versetzeinheit in  * ;
    :  !*   Arbeitsst. schwenken  * ;
    :  !*************************** ;
    :   ;
    :  LBL[51] ;
    :  R[41]=51    ;
    :  !FRG in Endlage halten ein ;
    :  DO[2165]=(ON) ;
    :  DO[2164]=(OFF) ;
    :  DO[2168]=(OFF) ;
    :  DO[18181]=(ON) ;
    :  WAIT (!DI[2165])    ;
    :  DO[18181]=(OFF) ;
    :  !Ueberwachungszeit Versetzeinheit ;
    :  TIMER[8]=((-5)) ;
    :  !Ueberwachungszeit Reinigung ;
    :  TIMER[9]=((-6)) ;
    :  !Versetzeinheit  in  Arbeitsst. ;
    :  DO[2168]=(!DI[2168] AND F[576]) ;
    :  IF (DO[2168] AND (TIMER[8]>=0) AND (DI[26] OR DI[27])),JMP LBL[51] ;
    :  IF ((DI[2168] AND F[576]) OR (!DI[2168] AND !F[576])),JMP LBL[52] ;
    :   ;
    :   ;
    :  !*************************** ;
    :  !*      Schritt 52         * ;
    :  !* MS1 Reinigung starten   * ;
    :  !*************************** ;
    :   ;
    :  LBL[52] ;
    :  R[41]=52    ;
    :  !MS1 Reinigung i.O. ;
    :  DO[18181]=(ON) ;
    :  WAIT (DI[1864])    ;
    :  DO[18181]=(OFF) ;
    :  !MS1 Ausblasen EIN ;
    :  DO[1870]=(ON) ;
    :  !MS1 Reinigung starten ;
    :  DO[1864]=(ON) ;
    :  !Einschaltdauer Reingung ;
    :  TIMER[7]=((R[26])) ;
    :  !IF (!DI[1864] AND (TIMER[9]>=0) ;
    :  DO[18181]=(ON) ;
    :  WAIT (!DI[1864])    ;
    :  WAIT ((TIMER[7]>=0))    ;
    :  DO[18181]=(OFF) ;
    :  !MS1 Reinigung beenden ;
    :  DO[1864]=(OFF) ;
    :  !MS1 Ausblasen AUS ;
    :  DO[1870]=(OFF) ;
    :  !MS1 Reinigung i.O. ;
    :  DO[18181]=(ON) ;
    :   ;
    :  WAIT (DI[1864])    ;
    :  DO[18181]=(OFF) ;
    :  !MS1 Einspruehen EIN ;
    :  DO[520]=(!F[574] AND F[575]) ;
    :  DO[1871]=(F[574] AND F[575]) ;
    :  !Einschaltdauer Einspruehen ;
    :  TIMER[7]=((R[23])) ;
    :  R[42]=52    ;
    :  JMP LBL[53] ;
    :   ;
    :  !**************************** ;
    :  !*        Schritt 53        * ;
    :  !*       MS1 Reinigung      * ;
    :  !*                          * ;
    :  !**************************** ;
    :   ;
    :  LBL[53] ;
    :  R[41]=53    ;
    :  !MS1 Reinigung (an Pneum. Schwenk ;
    :  F[323]=(OFF) ;
    :  DO[2163]=(OFF) ;
    :  DO[2164]=(OFF) ;
    :  DO[2165]=(OFF) ;
    :  DO[2166]=(OFF) ;
    :  DO[2168]=(OFF) ;
    :   ;
    :  !Ueberwachungszeit Schwenkeinheit ;
    :  TIMER[8]=((-7)) ;
    :  WAIT ((TIMER[7]>=0))    ;
    :  !MS1 Einspruehen AUS ;
    :  DO[520]=(OFF) ;
    :  DO[1871]=(OFF) ;
    :  !Versetzeinheit in Ruhest. schw. ;
    :  DO[2167]=(ON) ;
    :  DO[2168]=(OFF) ;
    :  !RSK Fehlerausgabe Schwenkeinheit ;
    :  F[324]=(!DI[2164]) ;
    :  !RSK Sammelstoerung ;
    :  F[329]=(F[324]) ;
